IF bEnable THEN
	// Alarm_0420	420	Error	Blokada podnośnika lub brak zasilania - sprawdź czujnik lub odblokuj mechanicznie
	//Error 1 - podnośnik nie porusza się pomimo wysterowania 
	tonErrorHeightChange(IN:=(bHeightMotorUp OR bHeightMotorDown) AND nLastPositionHeightCV=lrHeightMotorCV, PT:=T#3S);
	IF tonErrorHeightChange.Q THEN
		IF NOT arfbAlarm[0].bActive THEN
			bHeightMotorUp:=FALSE;
			bHeightMotorDown:=FALSE;
			arfbAlarm[0].Raise(nTimeStamp:=0);
		END_IF
	ELSE	
		IF  arfbAlarm[0].bActive AND bReset THEN
			arfbAlarm[0].Clear(nTimeStamp:=0, bResetConfirmation:= FALSE);
		END_IF	
// 		bHeightMotorUp:=FALSE;
// 		bHeightMotorDown:=FALSE;
// 		bError := TRUE;
// 		nErrorNr:=241;
// 		//nErrorNr := nErrorNr+iStationIndex;
// 		sErrorDescription:='Blokada podnośnika lub brak zasilania - sprawdź czujnik lub odblokuj mechanicznie';	
	END_IF
	// Alarm_0421	421	Error	Wartość zadana wysokości jest większa od maksymalnej - zmień ustawienia w recepturze {0}
	//Error 7 - Bład nastaw max
	tonMaxHeight(IN:=nPositionHeightSV>lrMaxHeight AND NOT bHomingDone AND eState=E_Station.eStarting,PT:=T#0S);
	IF tonMaxHeight.Q THEN
		arfbAlarm[1].ipArguments.Clear() .AddLReal(lrMaxHeight);
		IF NOT arfbAlarm[1].bActive THEN
			bHeightMotorUp:=FALSE;
			bHeightMotorDown:=FALSE;
			arfbAlarm[1].Raise(nTimeStamp:=0);
		END_IF
	ELSE	
		IF  arfbAlarm[1].bActive AND bReset THEN
			arfbAlarm[1].Clear(nTimeStamp:=0, bResetConfirmation:= FALSE);
		END_IF	
// 		bHeightMotorUp:=FALSE;
// 		bHeightMotorDown:=FALSE;
// 		bError := TRUE;
// 		nErrorNr:=242;
// 		//nErrorNr := nErrorNr+iStationIndex;
// 		sErrorDescription:='Wartość zadana wysokości jest większa od maksymalnej - zmień ustawienia w recepturze';
// 		sErrorDescription2:=REAL_TO_STRING(LREAL_TO_INT(lrMaxHeight));
	END_IF
	// Alarm_0422	422	Error	Wartość zadana wysokości jest mniejsza od minimalnej - zmień ustawienia w recepturze {0}
	//Error 8 - Bład nastaw min
tonMinHeight(IN:=nPositionHeightSV<lrMinHeight AND NOT bHomingDone AND eState=E_Station.eStarting,PT:=T#0S);
IF tonMinHeight.Q AND NOT bStateError THEN
	arfbAlarm[2].ipArguments.Clear() .AddLReal(lrMinHeight);
		IF NOT arfbAlarm[2].bActive THEN
			bHeightMotorUp:=FALSE;
			bHeightMotorDown:=FALSE;
			arfbAlarm[2].Raise(nTimeStamp:=0);
		END_IF
	ELSE	
		IF  arfbAlarm[2].bActive AND bReset THEN
			arfbAlarm[2].Clear(nTimeStamp:=0, bResetConfirmation:= FALSE);
		END_IF	
	//	bHeightMotorUp:=FALSE;
	//	bHeightMotorDown:=FALSE;
	//	bError := TRUE;
	//	nErrorNr:=243;
	//	//nErrorNr := nErrorNr+iStationIndex;
	//	sErrorDescription:='Wartość zadana wysokości jest mniejsza od minimalnej - zmień ustawienia w recepturze';
	//	sErrorDescription2:=REAL_TO_STRING(LREAL_TO_INT(lrMinHeight));	
END_IF

ELSE
	bError := FALSE;
END_IF

	
//******************PRZEJŚCIE DO eERROR*****************************

IF bError AND NOT bStateError THEN
	IF eLastState = eRunning THEN
		bCycleNotDone := TRUE;
	END_IF
	eState := E_Station.eError;
END_IF

//****************WYŚWIETLANIE STATUSU BLEDU***********************

(*Wyświetlanie błedu na wyjściu*)
bError							:= FALSE;
FOR nAlarmNumerator := 0 TO 19 DO
	bError						:= bError OR arfbAlarm[nAlarmNumerator].bActive;
END_FOR

(*Przepisywanie nazwy stacji*)
sErrorStationName := WSTRING_TO_STRING(sStationName);

//Jezeli nie zbazowane to potrzebne bazowanie
IF NOT bHeightMotorEncoderHomed  THEN
	bHomingDone:=FALSE;
END_IF
END_ACTION

ACTION HeightMotor:
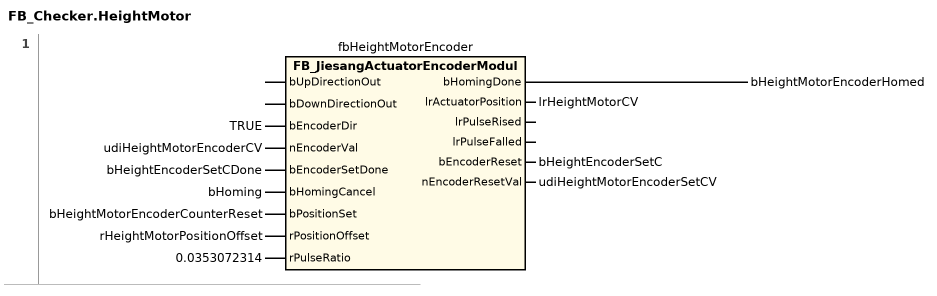
// NETWORK 1
fbHeightMotorEncoder(
    bEncoderDir := TRUE,
    nEncoderVal := udiHeightMotorEncoderCV,
    bEncoderSetDone := bHeightEncoderSetCDone,
    bHomingCancel := bHoming,
    bPositionSet := bHeightMotorEncoderCounterReset,
    rPositionOffset := rHeightMotorPositionOffset,
    rPulseRatio := 0.0353072314,
    lrActuatorPosition => lrHeightMotorCV,
    bEncoderReset => bHeightEncoderSetC,
    nEncoderResetVal => udiHeightMotorEncoderSetCV); // FB_JiesangActuatorEncoderModul
bHeightMotorEncoderHomed := fbHeightMotorEncoder.bHomingDone;
END_ACTION

ACTION Homing:
//BAZOWANIE

tofHeightMotorDown(IN:=bHeightMotorDown, PT:=T#1S); //Zabezpieczenie przed zbyt szybkim przełączeniem pomiędzy Down a Up, bezpiecznieki sie palą
	
//Podnoszenie stacji do maksymalnej pozycji
IF NOT bHeightMotorEncoderHomed OR rtEncoderHomed.Q THEN
	bHeightMotorUp:=(*TRUE*) NOT tofHeightMotorDown.Q;;
	bHeightMotorDown:=FALSE;
	IF tonHeightNoChange.Q THEN
		bHeightMotorEncoderCounterReset:=TRUE;
		bHeightMotorUp:=FALSE;
    END_IF
	//Jesli enkoder zbazowany zakończ bazowanie	
	IF rtEncoderHomed.Q THEN
		bHeightMotorUp:=FALSE;
		bHeightMotorDown:=FALSE;
		eState:=E_Station.eHomingDone;
	END_IF		
		
//Po podniesieniu stacji opuszczanie do ustalonej wysokości
ELSIF bHeightMotorEncoderHomed THEN
	bHeightMotorEncoderCounterReset:=FALSE;
	bHeightMotorUp:=lrHeightMotorCV<=nPositionHeightSV;
	bHeightMotorDown:=lrHeightMotorCV>=nPositionHeightSV;
	//Kiedy stacja osiągnie wysokość zadaną
	IF ABS(lrHeightMotorCV-nPositionHeightSV)<0.4 OR tonLimitPosMaxReachedDelay.Q OR tonLimitPosMinReachedDelay.Q THEN
		bHeightMotorDown:=FALSE;
		bHeightMotorUp:=FALSE;
		eState:=E_Station.eHomingDone;
	END_IF			
END_IF
END_ACTION

ACTION ManualMovements:

//W trybie ruchów manualnych wykonuj ruchy za pomocą rozkazów manualnych
IF NOT bRun THEN
	
	bHeightMotorUp:=bManualHeightMotorUp;
	bHeightMotorDown:=bManualHeightMotorDown;
ELSE	//Kasuje zeby po cyklu nic sie nie poruszało

	bManualHeightMotorUp  := FALSE;
	bManualHeightMotorDown  := FALSE;
END_IF


IF bHoming OR bHeightSet THEN
	eState:=E_Station.eHoming;
END_IF
	
Running();
	
//Zabezpieczenie przed kolizją stacji poprzez ruch podnośnika	
IF bHeightMotorDown AND lrHeightMotorCV<=lrMinHeight AND NOT bHoming AND NOT bHeightSet THEN
	bHeightMotorDown:=FALSE;
END_IF	

IF bHeightMotorUp AND lrHeightMotorCV>=lrMaxHeight AND NOT bHoming AND NOT bHeightSet THEN
	bHeightMotorUp:=FALSE;
END_IF
END_ACTION

ACTION Running:

//Timery
tofMotorUpPermition(IN:=bHeightMotorDown,PT:=T#250MS);
tofMotorDownPermition(IN:=bHeightMotorUp ,PT:=T#250MS);
tonOutputState(IN:=eRunningState=E_CheckerState.eFormPresent OR
				eRunningState=E_CheckerState.eBottleOK  OR
				eRunningState=E_CheckerState.eLidOK	 OR
				eRunningState=E_CheckerState.eCapOK OR
				eRunningState=E_CheckerState.eCapNOK
				,PT:=T#10MS);

CASE eRunningState OF
	
	E_CheckerState.eDisabled:
			eRunningState:=E_CheckerState.eReady;

	
	//SPRAWDZANIEGOTOWY DO PRACY
	E_CheckerState.eReady:
		//Jeśli wykryto czujnik formatki przejdź do stanu zasysania platynki
		IF bFormSensor THEN
			eRunningState:=E_CheckerState.eFormPresent;	
		END_IF

	//WYKRYTO FORMATKĘ
	E_CheckerState.eFormPresent:
		//Wykryto formatkę
		IF bBottleSensor THEN
			eRunningState:=E_CheckerState.eBottleOK;
		ELSIF bLidSensor THEN
			eRunningState:=E_CheckerState.eLidOK;
		ELSIF NOT bWenglorSensor THEN
			IF bCapSensor THEN
				eRunningState:=E_CheckerState.eCapOK;
			END_IF
		ELSIF bWenglorSensor THEN
			IF	bWenglorCapOk THEN
				eRunningState:=E_CheckerState.eCapOK;
			END_IF	
		ELSIF bCapNOKSensor THEN
			eRunningState:=E_CheckerState.eCapNOK;
		END_IF
		IF NOT bFormSensor THEN
			eRunningState:=E_CheckerState.eReady;
		END_IF

	//BUTELKA W FORMATCE
	E_CheckerState.eBottleOK:
		IF NOT bFormSensor THEN
			eRunningState:=E_CheckerState.eReady;
		END_IF
	
	//PLATYNKA OK
	E_CheckerState.eLidOK:
		IF NOT bFormSensor THEN
			eRunningState:=E_CheckerState.eReady;
		END_IF
	
	//NASADKA OK
	E_CheckerState.eCapOK:
		IF bCapNOKSensor THEN
			eRunningState:=E_CheckerState.eCapNOK;
		END_IF
		IF NOT bFormSensor THEN
			eRunningState:=E_CheckerState.eReady;
		END_IF	
		
		
	//NASADKA NOK
	E_CheckerState.eCapNOK:
		IF NOT bFormSensor THEN
			eRunningState:=E_CheckerState.eReady;
		END_IF			

END_CASE
END_ACTION

ACTION Statistics:

rtrigCycleTimerRead(CLK:=eRunningState=E_CheckerState.eFormPresent);
IF rtrigCycleTimerRead.Q THEN
		tCycleTime:=tonCycleTimer.ET;
END_IF
tonCycleTimer(IN:=eState>E_Station.eReady,PT:=T#1D);
END_ACTION

END_FUNCTION_BLOCK

// ---- POUs/FB/FB_VisionChecker_new.TcPOU
(*
Nazwa:			FB_VisionChecker
Opis:			stacja sprawdzania platynek czujnikiem wizyjnym
Wersja:			v1.0
Data:			2023-05-30
Autor:			DP
Urzadzenia:		Czujnik wizyjny KEYENCE
Konfiguracja:	
Info:
- 
*)

FUNCTION_BLOCK FB_VisionChecker_new
VAR_INPUT
	bEnable:BOOL;				//Zezowlenie na pracę stacji sprawdzania
	bEStop:BOOL;				//Stop Awaryjny nieaktywny
	bRun:BOOL;					//Rozkaz łapania 	
	bHoming:BOOL;				//Zezwolenie na wykonanie bazowania i pozycjonowania stacji sprawdzania
//	bHeightSet:BOOL;			//Ustaw wysokość
	bIgnoreError:BOOL;			//Ignorowania błędów cyklu pracy
	bReset:BOOL;				//Reset błędu, jeśli w stanie "eError"
//	nPositionHeightSV:LREAL;	//Wysokość zadana na której ma znajdować się stacja sprawdzania
	bManualMovement:BOOL; 		//Uruchomienie trybu ruchów ręcznych
//	lrMaxHeight:LREAL;			//Maksymalna wysokość stacji sprawdzania
//	lrMinHeight:LREAL;			//Minimalna wysokość stacji sprawdzania
	uiCameraActualProgram:UINT;
	iCameraSetProgram:INT;
	bCameraError:BOOL; 
	bCameraGood:BOOL; 	
	bCameraLogic1CapPresent:BOOL; 		
	bCameraBusy:BOOL; 	
	//StepMode
//	bStepMode				: BOOL;		//Włączony tryb skokowy sterowania podnośnikami (tylko w serwisie)
//	lrSetPosStepMode		: LREAL; 	//Ruch podnośnika o zadaną wartość w trybie krokowym (tylko w serwisie)
	
//	_HEIGHTMOTOR_ :BOOL;	
//	bHeightMotorEncoderPulse :BOOL;			//Sygnał impulsów enkodera siłownika
//	rHeightMotorPositionOffset :REAL;		//Wysokość bazowani podnośnika

	_ALARMINFO_ :BOOL;
	iStationIndex:UDINT;					//Numer stacji 
	sStationName:STRING;					//Nazwa stacji	

END_VAR
VAR_OUTPUT	
	eState: E_Station;						//Stan ogólny bloku
	eRunningState: E_CheckerState;			//Stan stacji sprawdzania
	bError: BOOL;							//Błąd stacji
	nErrorNr: UDINT;						//Nr błędu stacji sprawdzania
	sErrorDescription:STRING(200);			//Opis błędu
	sErrorDescription2:STRING(200);			//Opis błędu
	sErrorStationName:STRING;				//Nazwa stacji
	udiStationID: UDINT;				// Nr stacji

//	bHeightMotorUp:BOOL;					//Sterowanie silnikiem podnośnika  - RUCH W GÓRĘ
//	bHeightMotorDown:BOOL;					//Sterowanie silnikiem podnośnika  - RUCH W DÓŁ
//	lrHeightMotorCV:LREAL;					//Aktualna wysokość stacji sprawdzania
	bCameraTrigger:BOOL; 
	uiCameraProgram:UINT; 
	bCameraChangeProgram:BOOL; 	
	bCheckOK:BOOL;							//Platynka OK
	bCapPresent:BOOL;
	tCycleTime:TIME;	
	bHomingDone:BOOL;						//Wymagane ponowne bazowanie (blad podczas bazowania lub stop awaryjny)
	bCycleDone:BOOL;
	bCycleNotDone:BOOL;
	AsProgramDescription: ARRAY [0..10] OF STRING;	// Opis programów

END_VAR
VAR
//	tonHeightNoChange: TON; // Timer wykrycia braku ruchu siłownika zmiany wysokości stacji
//	nLastPositionHeightCV: LREAL;// Pozycja podnośnika w poprzednim cyklu programu
//	tonErrorHeightChange: TON; // Timer błędu podnośnika
	rtEncoderHomed:R_TRIG;
	tonCycleTimer:TON;
	rtrigCycleTimerRead:R_TRIG;
	tonTriggerDelay: TON;
	tonNotBusyDelay: TON;
	tonLidNOK: TON;
	tofMotorUpPermition: TOF;
	tofMotorDownPermition: TOF;
	tonLimitPosMinReachedDelay: TON;
	tonLimitPosMaxReachedDelay: TON;
	tonMaxHeight: TON;
	tonMinHeight: TON;
	
	//Podnośnik Jiesang	
	fbHeightMotorEncoder: FB_JiesangActuatorEncoder_1;	// Blok enkodera podnośnika chwytaka stabilizującego pod zakręcarką	
	bHeightMotorEncoderCounterReset:BOOL; 				// Sygnał resetu enkodera
	bHeightMotorEncoderHomed:BOOL;						// Informacja od enkodera że jest zbazowany

	eLastState: E_Station;								// Stan ogólny bloku
	eLastRunningState: E_CheckerState;					// Stan podbloku
	eLastStateTemp: E_Station;							// Stan ogólny bloku
	eLastRunningStateTemp: E_CheckerState;				// Stan podbloku	
	
	bStateError: BOOL;

	//Step Mode
	rtStepModeUp			: R_TRIG;
	rtStepModeDown			: R_TRIG;
	lrStepModeHeightMotorSV	: LREAL;
	bStepModeMoving			: BOOL;
	tofStepModeMoving		: TOF;	
	rtCheckingEnd			: R_TRIG;
	tonbCameraChangeProgram: TON;
	rtuiCameraActualProgram: R_TRIG;
	tonTryChangeProgram: TON;
END_VAR

//HeightMotor();
ErrorHandling();
Control();
Statistics();
Programs();
aStationID();

(*Zapisywanie ostatniego stanu*)
IF eLastStateTemp<>eState THEN
	eLastState := eLastStateTemp;
END_IF
eLastStateTemp := eState;
IF eLastRunningStateTemp<>eRunningState THEN
	eLastRunningState := eLastRunningStateTemp;
END_IF
eLastRunningStateTemp := eRunningState;
(*Koniec Zapisywanie ostatniego stanu*)

//nLastPositionHeightCV:=lrHeightMotorCV;

ACTION aStationID:
udiStationID	:=	iStationIndex;
END_ACTION

ACTION Control:

	(** TIMERY**)
	rtEncoderHomed				(CLK:=bHeightMotorEncoderHomed,																Q=>);


	(*****Wyłączenie enable*****)
	IF NOT bEnable THEN
		IF eState <> E_Station.eDisabled AND eState <> E_Station.ePreparingToDisable THEN
				eState 							:=	E_Station.ePreparingToDisable; 
		END_IF	
	END_IF

	(*****Estop*****)
	IF NOT bEstop  THEN	
		IF eState <> E_Station.eAborted AND eState <> E_Station.eAborting AND eState <> E_Station.eDisabled THEN
				eState 							:=	E_Station.eAborting; 
		END_IF
	END_IF

	
	CASE eState OF
	/////////////////////////////	
		E_Station.eDisabled: 					// Stan nieaktywnosci (Stacja wyłączona) 
		
			IF bEnable THEN
				eState 							:=	E_Station.ePreparingToReady; 
			END_IF 
			
    /////////////////////////////	    
		E_Station.eAborted: 					// Stan bezpiecznego zatrzymania (po Abortingu) 

			IF bEStop THEN
				eState 							:=	E_Station.ePreparingToReady;
			END_IF
			
	/////////////////////////////	
		E_Station.eAborting:                 	// Stan bezpiecznego zatrzymywania (po EStopie)
			
//			bHeightMotorUp						:=	FALSE;
//			bHeightMotorDown					:=	FALSE;
			eState 								:=	E_Station.eAborted;  
			eRunningState						:=	E_CheckerState.eDisabled;
			
	/////////////////////////////			
		E_Station.eError:                 	 	// Stan błędu 	
	
			IF bReset THEN
				eState 							:=	E_Station.eResetting;
			ELSE
				ResetCommands();
			END_IF
			
	/////////////////////////////
		E_Station.eResetting:					// Stan resetowania bledu (po Errorze)
			
			bError := FALSE;
			IF NOT bError THEN
				nErrorNr 						:=	0;
   				sErrorDescription 				:=	'';
				eState 							:=	E_Station.ePreparingToReady;
			ELSE
				eState 							:=	E_Station.eError;
			END_IF
        
	/////////////////////////////
		E_Station.eManualMovement:     			// Stan ruchów manualnych  
       
			ManualMovements();
			//Wyjście z trybu serwisowego
//			IF NOT bManualMovement THEN
//				bHeightMotorUp					:=	FALSE;
//				bHeightMotorDown				:=	FALSE;	
//				eState							:=	E_Station.eReady;
//			END_IF

	/////////////////////////////
		E_Station.eHoming:						// Stan bazowania 

			Homing();
//			IF NOT bHoming AND NOT bHeightSet THEN
//				bHeightMotorDown				:=	FALSE;
//				bHeightMotorUp					:=	FALSE;
				eState							:=	E_Station.ePreparingToReady;
//			END_IF		
			
	/////////////////////////////
		E_Station.eHomingDone:                  // Stan wykonania bazowania 
		
//			bHeightMotorDown					:=	FALSE;
//			bHeightMotorUp						:=	FALSE;
//			bHeightMotorEncoderCounterReset		:=	FALSE;
			bHomingDone							:=	TRUE;
//			IF NOT bHoming AND NOT bHeightSet THEN
			   eState							:=	E_Station.eReady;
//			END_IF
			
	/////////////////////////////
		E_Station.ePreparingToReady:            // Stan przygotowywania do gotowosci (zawsze przed Ready)  
		
			eRunningState						:=	E_CheckerState.eReady;
			eState								:=	E_Station.eReady;	
			
	/////////////////////////////
		E_Station.ePreparingToDisable:          // Stan przygotowywania do nieaktywnosci (po wyłączeniu Enable) 
  
//			bHeightMotorUp						:=	TRUE;
//			bHeightMotorDown					:=	FALSE;	
//			IF tonHeightNoChange.Q THEN
//				bHeightMotorUp					:=	FALSE;
				eState							:=	E_Station.eDisabled;
				eRunningState					:=	E_CheckerState.eDisabled;
//			END_IF	
				
	/////////////////////////////
		E_Station.eReady:						// Stan gotowosci 
			
			IF bRun AND NOT bCycleDone AND NOT bCycleNotDone THEN
				eState 							:=	E_Station.eStarting; 
			END_IF
			IF bHoming (*OR bHeightSet*) THEN
				eState 							:=	E_Station.eHoming; 
			END_IF
			IF bManualMovement THEN
				//Jeśli przejście w tryb ruchów manualnych przepisz wszystkie stany siłowników sterowanych przez moduł
				//aby zapobiec ewentualnym kolizjom po wejściu w tryb serwisowy
//				bManualHeightMotorUp			:=	bHeightMotorUp;
//				bManualHeightMotorDown			:=	bHeightMotorDown;
				eState 							:=	E_Station.eManualMovement; 
			END_IF
			IF NOT bRun THEN
				bCycleDone 						:=	FALSE;
				bCycleNotDone 					:=	FALSE;			
			END_IF
			
	/////////////////////////////
		E_Station.eStopping:					// Stan zatrzymywania 
			
			Running();
			bCameraTrigger						:= FALSE;
			bCheckOK							:= FALSE;
			eState								:=	E_Station.eReady;
			
	/////////////////////////////
		E_Station.eStarting:                  	// Stan uruchamiania (po Ready)
		
			eRunningState						:= E_CheckerState.eReady;
			eState								:= E_Station.eRunning; 

	/////////////////////////////
		E_Station.eRunning:               		// Stan wykonywania cyklu (po Startingu), w tym stanie osobny
 
			Running();
			IF NOT bRun THEN 					(*Przerywanie cyklu*)
				eState							:=	E_Station.eStopping;
				bCycleNotDone					:=	TRUE;
			END_IF
			(*IF bCycleDone OR bCycleNotDone THEN (*Cykl zakończony*)
				eState 				 := E_Station.eReady;
			END_IF*)						
			
	/////////////////////////////		
	END_CASE
END_ACTION

ACTION ErrorHandling:
//OBSŁUGA BŁĘDÓW STACJI SPRAWDZANIA

//************LISTA BŁĘDÓW***************
bStateError:= (eState=E_Station.eError) OR (eState=E_Station.eResetting) OR bIgnoreError;

IF bEnable THEN

//	//Error 1 - podnośnik nie porusza się pomimo wysterowania 
//	tonErrorHeightChange(IN:=(bHeightMotorUp OR bHeightMotorDown) AND nLastPositionHeightCV=lrHeightMotorCV, PT:=T#3S);
//	IF tonErrorHeightChange.Q AND NOT bStateError THEN
//		bHeightMotorUp:=FALSE;
//		bHeightMotorDown:=FALSE;
//		bError := TRUE;
//		nErrorNr:=301;
//		//nErrorNr := nErrorNr+iStationIndex;
//		sErrorDescription:='Blokada podnośnika lub brak zasilania - sprawdź czujnik lub odblokuj mechanicznie';	
//	END_IF
	
//	//Error 2 - Bład nastaw max
//	tonMaxHeight(IN:=nPositionHeightSV>lrMaxHeight AND NOT bHomingDone AND eState=E_Station.eStarting,PT:=T#0S);
//	IF tonMaxHeight.Q AND NOT bStateError THEN
//		bHeightMotorUp:=FALSE;
//		bHeightMotorDown:=FALSE;
//		bError := TRUE;
//		nErrorNr:=302;
//		//nErrorNr := nErrorNr+iStationIndex;
//		sErrorDescription:='Wartość zadana wysokości jest większa od maksymalnej - zmień ustawienia w recepturze';
//		sErrorDescription2:=REAL_TO_STRING(LREAL_TO_INT(lrMaxHeight));
//	END_IF
	
	//Error 3 - Bład nastaw min
	//tonMinHeight(IN:=nPositionHeightSV<lrMinHeight AND NOT bHomingDone AND eState=E_Station.eStarting,PT:=T#0S);
	//IF tonMinHeight.Q AND NOT bStateError THEN
	//	bHeightMotorUp:=FALSE;
	//	bHeightMotorDown:=FALSE;
	//	bError := TRUE;
	//	nErrorNr:=303;
	//	//nErrorNr := nErrorNr+iStationIndex;
	//	sErrorDescription:='Wartość zadana wysokości jest mniejsza od minimalnej - zmień ustawienia w recepturze';
	//	sErrorDescription2:=REAL_TO_STRING(LREAL_TO_INT(lrMinHeight));	
	//END_IF

ELSE
	bError := FALSE;
END_IF

	
//******************PRZEJŚCIE DO eERROR*****************************

IF bError AND NOT bStateError THEN
	IF eLastState = eRunning THEN
		bCycleNotDone := TRUE;
	END_IF
	eState := E_Station.eError;
END_IF

//****************WYŚWIETLANIE STATUSU BLEDU***********************

(*Wyświetlanie błedu na wyjściu*)
bError;

(*Przepisywanie nazwy stacji*)
sErrorStationName := sStationName;

//Jezeli nie zbazowane to potrzebne bazowanie
IF NOT bHeightMotorEncoderHomed  THEN
	bHomingDone:=FALSE;
END_IF
END_ACTION

ACTION Homing:
//BAZOWANIE
eState:=E_Station.eHomingDone;
	
////Podnoszenie stacji do maksymalnej pozycji
//IF NOT bHeightMotorEncoderHomed OR rtEncoderHomed.Q THEN
//	bHeightMotorUp:=TRUE;
//	bHeightMotorDown:=FALSE;
//	IF tonHeightNoChange.Q THEN
//		bHeightMotorEncoderCounterReset:=TRUE;
//		bHeightMotorUp:=FALSE;
//    END_IF
//	//Jesli enkoder zbazowany zakończ bazowanie	
//	IF rtEncoderHomed.Q THEN
//		bHeightMotorUp:=FALSE;
//		bHeightMotorDown:=FALSE;
//		eState:=E_Station.eHomingDone;
//	END_IF		
		
////Po podniesieniu stacji opuszczanie do ustalonej wysokości
//ELSIF bHeightMotorEncoderHomed THEN
//	bHeightMotorEncoderCounterReset:=FALSE;
//	bHeightMotorUp:=lrHeightMotorCV<=nPositionHeightSV;
//	bHeightMotorDown:=lrHeightMotorCV>=nPositionHeightSV;
//	//Kiedy stacja osiągnie wysokość zadaną
//	IF ABS(lrHeightMotorCV-nPositionHeightSV)<1 OR tonLimitPosMaxReachedDelay.Q OR tonLimitPosMinReachedDelay.Q THEN
//		bHeightMotorDown:=FALSE;
//		bHeightMotorUp:=FALSE;
//		eState:=E_Station.eHomingDone;
//	END_IF			
//END_IF
END_ACTION

ACTION ManualMovements:

//W trybie ruchów manualnych wykonuj ruchy za pomocą rozkazów manualnych
IF NOT bRun THEN
	eRunningState		:=	E_CheckerState.eReady;
	bCameraTrigger		:=	FALSE;
	bCheckOK			:=	FALSE;
//	bHeightMotorUp		:=	bManualHeightMotorUp;
//	bHeightMotorDown	:=	bManualHeightMotorDown;
ELSE	//Kasuje zeby po cyklu nic sie nie poruszało
//	bManualHeightMotorUp  := FALSE;
//	bManualHeightMotorDown  := FALSE;
END_IF


IF bHoming (*OR bHeightSet*) THEN
	eState:=E_Station.eHoming;
END_IF
	
Running();

	
//Zabezpieczenie przed kolizją stacji poprzez ruch podnośnika	
//IF bHeightMotorDown AND lrHeightMotorCV<=lrMinHeight AND NOT bHoming AND NOT bHeightSet THEN
//	bHeightMotorDown:=FALSE;
//END_IF	

//IF bHeightMotorUp AND lrHeightMotorCV>=lrMaxHeight AND NOT bHoming AND NOT bHeightSet THEN
//	bHeightMotorUp:=FALSE;
//END_IF
END_ACTION

ACTION Programs:
tonbCameraChangeProgram	(IN:=bCameraChangeProgram,PT:=T#1S);
tonTryChangeProgram	(IN:=uiCameraActualProgram <> uiCameraProgram AND NOT bCameraChangeProgram, PT:=T#5S);
rtuiCameraActualProgram	(CLK:=uiCameraActualProgram <> uiCameraProgram,	Q=>);
uiCameraProgram	:=	INT_TO_UINT(iCameraSetProgram);

IF rtuiCameraActualProgram.Q	 OR  tonTryChangeProgram.Q THEN
	bCameraChangeProgram	:=	TRUE;
END_IF
IF tonbCameraChangeProgram.Q THEN
	bCameraChangeProgram	:=	FALSE;
END_IF

(*Narzędzia*)
AsProgramDescription[0] := '1. opak:butelka płaska, nasadka:wbijana biała';
AsProgramDescription[1] := '2. opak:rezerwa, nasadka:rezerwa';
AsProgramDescription[2] := '3. opak:rezerwa, nasadka:rezerwa';
AsProgramDescription[3] := '4. opak:rezerwa, nasadka:rezerwa';
AsProgramDescription[4] := '5. opak:rezerwa, nasadka:rezerwa';
AsProgramDescription[5] := '6. opak:rezerwa, nasadka:rezerwa';
AsProgramDescription[6] := '7. opak:rezerwa, nasadka:rezerwa';
AsProgramDescription[7] := '8. opak:rezerwa, nasadka:rezerwa';
AsProgramDescription[8] := '9. opak:rezerwa, nasadka:rezerwa';
AsProgramDescription[9] := '10. opak:rezerwa, nasadka:rezerwa';
AsProgramDescription[10] := '11. opak:rezerwa, nasadka:rezerwa';
END_ACTION

ACTION ResetCommands:

//bStepModeMoving 			:= FALSE;
//bHeightMotorDown			:= FALSE;
//bHeightMotorUp				:= FALSE;
//bManualHeightMotorUp		:= FALSE;
//bManualHeightMotorDown		:= FALSE;
END_ACTION

ACTION Running:

//Timery
//tofMotorUpPermition		(IN:=	bHeightMotorDown,								PT:=T#250MS);
//tofMotorDownPermition	(IN:=	bHeightMotorUp,									PT:=T#250MS);
tonTriggerDelay			(IN:=	eRunningState=E_CheckerState.eFormPresent,		PT:=T#50MS);//bylo 50
tonNotBusyDelay			(IN:=	tonTriggerDelay.Q AND NOT bCameraBusy,
																				PT:=T#50MS);
tonLidNOK				(IN:=	eRunningState=E_CheckerState.eFormPresent,
																				PT:=T#50MS);				

CASE eRunningState OF
	
	E_CheckerState.eDisabled:
	
		eRunningState		:=	E_CheckerState.eReady;
	
	//SPRAWDZANIEGOTOWY DO PRACY
	E_CheckerState.eReady:
		
		IF bRun THEN
			eRunningState	:=	E_CheckerState.eFormPresent;	
		END_IF

	//WYKRYTO SLOIK
	E_CheckerState.eFormPresent:
	
		bCameraTrigger		:= TRUE;
		IF	tonTriggerDelay.Q THEN
			IF tonNotBusyDelay.Q AND bCameraGood THEN
				eRunningState	:=	E_CheckerState.eLidOK;		
			ELSIF tonNotBusyDelay.Q  THEN
				eRunningState	:=	E_CheckerState.eLidNOK;	
			END_IF	
		END_IF
		
	
	//BUTELKA W FORMATCE
	E_CheckerState.eBottleOK:
	;
	
	//PLATYNKA OK
	E_CheckerState.eLidOK:
	
		bCheckOK	:= TRUE;
		bCycleDone	:= TRUE;
		bCapPresent	:= bCameraLogic1CapPresent;	
	
	//PLATYNKA NOK
	E_CheckerState.eLidNOK:

		bCheckOK	:= FALSE;	
		bCycleDone	:= TRUE;
		bCapPresent	:= bCameraLogic1CapPresent;
		
	//NASADKA OK
	E_CheckerState.eCapOK:
	;
		
	//NASADKA NOK
	E_CheckerState.eCapNOK:
	;		

	E_CheckerState.eChecking:
	;
		
END_CASE
END_ACTION

ACTION Statistics:

rtrigCycleTimerRead(CLK:=eRunningState=E_CheckerState.eLidOK OR eRunningState=E_CheckerState.eLidNOK);
IF rtrigCycleTimerRead.Q THEN
		tCycleTime:=tonCycleTimer.ET;
END_IF
tonCycleTimer(IN:=eState>E_Station.eReady,PT:=T#1D);
END_ACTION

END_FUNCTION_BLOCK

// ---- POUs/FB/Various/FB_Average.TcPOU
(********************************************************************************************)
(*							Beckhoff Automation Poland										*)
(*								FB_Average	 v1.2											*)
(*									2.02.2011												*)
(*								v1.2 Optymalizacja wewnętrzna								*)
(*					Blok funkcyjny obliczający średnią z wartości wejściowej rValue			*)
(*					w zadanym przedziale czasowym lub z określonej ilości pomiarów			*)
(*__________________________________________________________________________________________*)
FUNCTION_BLOCK FB_Average
VAR_INPUT
	rValue : 			REAL;			(*Uśredniana wartość*)
	tInterval : 		TIME;			(*Co jaki czas ma byc robiony wpis*)
END_VAR
VAR_OUTPUT
	rAverage: 			REAL; 			(*Wartość średnia*)
END_VAR
VAR CONSTANT
	MAX_INDEX: 			USINT 	:= 10 ;	(*Ilość wpisów do uśredniania*)
END_VAR
VAR
	aData: 				ARRAY[0..MAX_INDEX] OF REAL;
	nIndex:		 		USINT;			(*Ostatni wpis, czyli przyjmuje wartosci od 0 do MAX_INDEX - 1*)
	i:					USINT;			(*Iterator*)
	ttimer: 			TON;
	suma: 				REAL;
END_VAR

ttimer(IN:= NOT ttimer.Q, PT:= tInterval, Q=> , ET=> );

IF nIndex = 0 THEN	(*Na poczatku wypelniamy pierwsza komorke w tablicy*)
	nIndex := 1;
	aData[0] := rValue;
END_IF

IF ttimer.Q THEN
	suma := 0;
	FOR i := 1 TO nIndex DO
		aData[i - 1] := aData[i];
		suma := suma + aData[i];
	END_FOR
	IF	nIndex < (MAX_INDEX) THEN
		nIndex := nIndex + 1;
	END_IF
	aData[nIndex] := rValue;
END_IF

rAverage := suma/nIndex;

END_FUNCTION_BLOCK

// ---- POUs/P09_CapPuttedCheck.TcPOU
(*
Nazwa:			P09_CapPuttedCheck
Opis:			Stacja sprawdzania nasadek
Wersja:			v0.1
Data:			2018-10-10
Autor:			DP
Urzadzenia:		
Konfiguracja:	
Info:

*)
PROGRAM P09_CapPuttedCheck
VAR_INPUT
	IbCapPuttedCheckSensor 				AT %I*		:BOOL;		// Wejście wykrycia nasadki 
	IbCapPuttedCheckFormSensor 			AT %I*		:BOOL;		// Wejście wykrycia formatek w sprawdzaniu nasadek
END_VAR
VAR
	fbCapPuttedCheck								:FB_Checker;
	eCapPuttedCheckState							:E_Station; 			// Stan pracy podajnika platynek			
	eCapPuttedCheckRunningState						:E_CheckerState; 		// Stan pracy podajnika platynek
	fbCapPuttedCheckState							:FB_State;
	
	IbCapPuttedCheckHeightEncoderPulses				AT %I*:BOOL;		//	(*PLC.A14*) 	// Enkoder podnośnika czujnika kontroli nakrętki
	QbCapPuttedCheckHeightUpCmd 					AT %Q*: BOOL; 				//	(*PLC.A19*) 	// Wyjście sterujące podnośnikiem sprawdzania nasadek w formatkach, Silnik w górę
	QbCapPuttedCheckHeightDownCmd 					AT %Q*: BOOL; 			//	(*PLC.A19*)		// Wyjście sterujące podnośnikiem sprawdzania nasadek w formatkach, Silnik w dół
	IbCapPuttedCheckWenglorFormSensor				AT %I*:BOOL;
	fbIbCapPuttedCheckFormSensor					:FB_InputFilter; //Wejście przefiltrowane czujnika

	IbCapPuttedCheckEncoderSetCDone				AT %I*: BOOL;	
    IudiCapPuttedCheckHeightEncoderCV          AT %I*: UDINT;
    QbCapPuttedCheckHeightEncoderSetC 			AT %Q*: BOOL;
    QudiCapPuttedCheckHeightEncoderSetCV       AT %Q*: UDINT;
	
	TimerCapPuttedCheckEnable						: TOF;
	tonCapPuttedCheckEnable							: TON;		
	rtEnable										: R_TRIG;
	tonCapPuttedFormsCheckRFID						: TON;
	rtCapPuttedFormCheck							: R_TRIG;

	tonStoppingCapPuttedTooLong: TON;
	IdiCapPuttedCheckSensorCV_Wenglor					AT %I*:DINT;
	IbCapPuttedCheckSensorScale_Wenglor					AT %I*:BYTE;
	IbCapPuttedCheckSensorWarning_1_Wenglor				AT %I*:BOOL;
	IbCapPuttedCheckSensorWarning_2_Wenglor				AT %I*:BOOL;	
	IbCapPuttedCheckSensorWarning_3_Wenglor				AT %I*:BOOL;
	IbCapPuttedCheckSensorWarning_4_Wenglor				AT %I*:BOOL;
	IbCapPuttedCheckSensorWarning_Wenglor				AT %I*:BOOL;
	IbCapPuttedCheckSensorError_Wenglor                	AT %I*:BOOL;
	IbCapPuttedCheckSensorSSC1_Wenglor                 	AT %I*:BOOL;
	IbCapPuttedCheckSensorSSC2_Wenglor                 	AT %I*:BOOL;
	QbCapPuttedCheckSensorControlSignal_Wenglor			AT %Q*:BOOL;
	QbCapPuttedCheckSensorFindMe_Wenglor				AT %Q*:BOOL;
	QbCapPuttedCheckSensorTeachSSC1_Wenglor             AT %Q*:BOOL;
	QbCapPuttedCheckSensorTeachSSC2_Wenglor				AT %Q*:BOOL;
	
	bCapPuttedCheckSensorWenglorBottleTooFar	:BOOL;
	bCapPuttedCheckSensorWenglorBottleTooClose	:BOOL;
	bCapPuttedCheckSensorWenglorNoData	:BOOL;
	diDistanceSensorToTransporter		:DINT;
	
	
	lrCapPuttedCheckSensorCV						: LREAL;
	lrCapPuttedCheckSensorFilteredCV				: LREAL;
	lrCapPuttedCheckSensorAveragedCV				: LREAL;	
	fbCapPuttedCheckSensorFilter					: FB_FilterEx;
	fbCapPuttedCheckSensorAverage					: FB_Average;	
	lrCapPuttedCheckSensorLimitLow: LREAL;
	lrCapPuttedCheckSensorLimitHigh: LREAL;
	bCapPuttedCheckSensorLimitOK: BOOL;
	bCapPuttedCheckSensorLimitNOK: BOOL;	
	tonCapPuttedCheckSensorLimitOK: TON;
	tonCapPuttedCheckSensorLimitNOK: TON;
	bCapPuttedCheckSensorShinyMode: BOOL;
	bCapPuttedCheckSensorPointedMode: BOOL;	
END_VAR



tonStoppingCapPuttedTooLong(IN:=P00_PackML.fbPMLAuto.ePMLState = E_PMLState.ePMLState_STOPPING,PT:=T#3S);
IF P00_PackML.fbPMLAuto.ePMLState = E_PMLState.ePMLState_EXECUTE OR P00_PackML.fbPMLAuto.ePMLState = E_PMLState.ePMLState_STARTING THEN
	bCapPuttedCheckRun:=TRUE;
ELSIF tonStoppingCapPuttedTooLong.Q THEN
	bCapPuttedCheckRun:=FALSE;
END_IF
aCapPuttedCheck();
aCapPuttedCheckSensor();

tonCapPuttedFormsCheckRFID(IN:=IbCapPuttedCheckFormSensor, PT:=T#25MS);//było 10
rtCapPuttedFormCheck(CLK:=tonCapPuttedFormsCheckRFID.Q);


fbIbCapPuttedCheckFormSensor(bIN:=IbCapPuttedCheckFormSensor, tFilterTimeOn:=T#10MS, tFilterTimeOff:=T#10MS);

(* BAZOWANIE - ZMIAN*)
tonCapPuttedCheckEnable(IN:=fbCapPuttedCheck.bEnable,PT:=T#5S); (*Dodany ton bo Wizka zjebnie wgrywa zmienne, najpierw włacza Enabla a potem dopiero wybiera recepture*)
rtEnable(CLK:=tonCapPuttedCheckEnable.Q,Q=>);

IF rtEnable.Q AND (P00_PackML.fbPMLAuto.ePMLState = E_PMLState.ePMLState_IDLE OR P00_PackML.fbPMLAuto.ePMLState = E_PMLState.ePMLState_EXECUTE)  THEN
		VIS.bCapPuttedCheckHeightSet											:= TRUE;
ELSIF fbCapPuttedCheck.eState=E_Station.eHomingDone  OR VIS.bErrorOccure THEN
 		VIS.bCapPuttedCheckHeightSet											:= FALSE;
END_IF

(*KONIEC BAZOWANIE - ZMIANA*)

(********* GENEROWANIE STANU STACJI DO WIZKI**********)
fbCapPuttedCheckState(
	eState																		:= eCapPuttedCheckState , 
	bRun																		:= P00_PackML.fbPMLAuto.ePMLState = E_PMLState.ePMLState_EXECUTE ,	
	eCheckerRunningState														:= eCapPuttedCheckRunningState , 
	sStateDesc																	=> VIS.sCapPuttedCheckState,
	iState																		=> VIS.iCapPuttedCheckState );
(***** KONIEC GENEROWANIE STANU STACJI DO WIZKI*******)	

(*Opoznienie wyłączanie enabla*)
TimerCapPuttedCheckEnable (IN:=bCapPuttedCheckEnable , PT:=T#2S);



(****WENGLOR*************)
lrCapPuttedCheckSensorLimitLow:=diDistanceSensorToTransporter-VIS.iPackageHeightShow;
lrCapPuttedCheckSensorLimitHigh:=diDistanceSensorToTransporter-VIS.iPackageHeightShow+150;

ACTION aCapPuttedCheck:
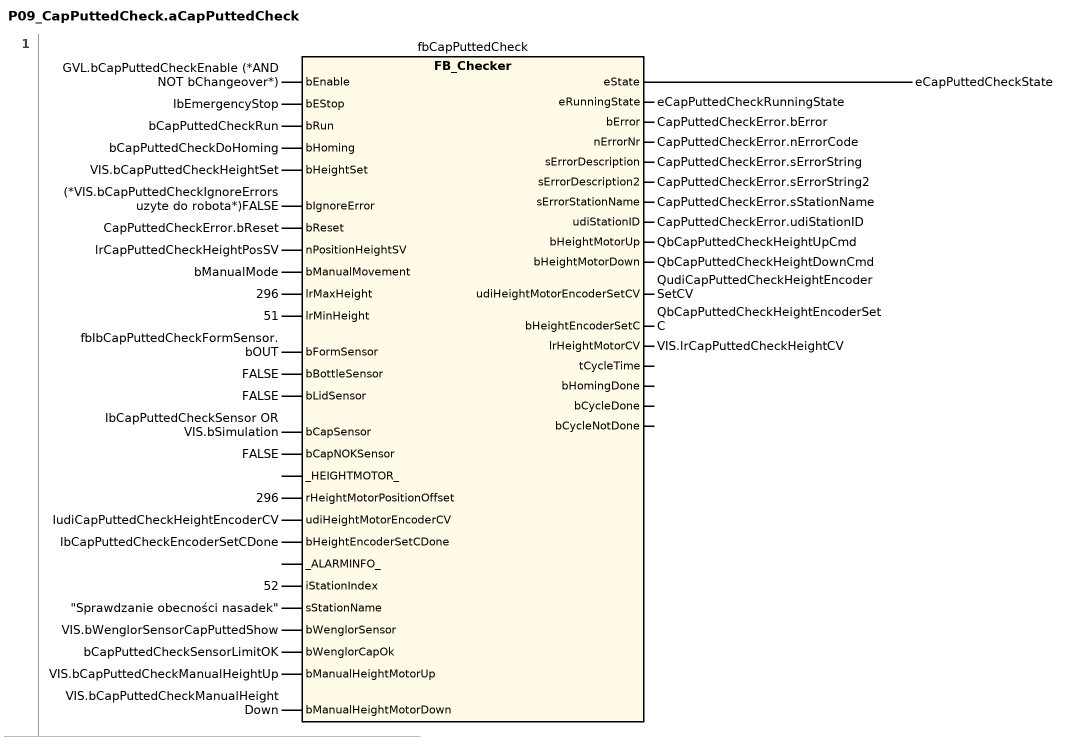
// NETWORK 1
fbCapPuttedCheck(
    bEnable := GVL.bCapPuttedCheckEnable (*AND NOT bChangeover*),
    bEStop := IbEmergencyStop,
    bRun := bCapPuttedCheckRun,
    bHoming := bCapPuttedCheckDoHoming,
    bHeightSet := VIS.bCapPuttedCheckHeightSet,
    bIgnoreError := (*VIS.bCapPuttedCheckIgnoreErrors uzyte do robota*)FALSE,
    bReset := CapPuttedCheckError.bReset,
    nPositionHeightSV := lrCapPuttedCheckHeightPosSV,
    bManualMovement := bManualMode,
    lrMaxHeight := 296,
    lrMinHeight := 51,
    bFormSensor := fbIbCapPuttedCheckFormSensor.bOUT,
    bBottleSensor := FALSE,
    bLidSensor := FALSE,
    bCapSensor := IbCapPuttedCheckSensor OR VIS.bSimulation,
    bCapNOKSensor := FALSE,
    rHeightMotorPositionOffset := 296,
    udiHeightMotorEncoderCV := IudiCapPuttedCheckHeightEncoderCV,
    bHeightEncoderSetCDone := IbCapPuttedCheckEncoderSetCDone,
    iStationIndex := 52,
    sStationName := "Sprawdzanie obecności nasadek",
    bWenglorSensor := VIS.bWenglorSensorCapPuttedShow,
    bWenglorCapOk := bCapPuttedCheckSensorLimitOK,
    bManualHeightMotorUp := VIS.bCapPuttedCheckManualHeightUp,
    bManualHeightMotorDown := VIS.bCapPuttedCheckManualHeightDown,
    eRunningState => eCapPuttedCheckRunningState,
    bError => CapPuttedCheckError.bError,
    nErrorNr => CapPuttedCheckError.nErrorCode,
    sErrorDescription => CapPuttedCheckError.sErrorString,
    sErrorDescription2 => CapPuttedCheckError.sErrorString2,
    sErrorStationName => CapPuttedCheckError.sStationName,
    udiStationID => CapPuttedCheckError.udiStationID,
    bHeightMotorUp => QbCapPuttedCheckHeightUpCmd,
    bHeightMotorDown => QbCapPuttedCheckHeightDownCmd,
    udiHeightMotorEncoderSetCV => QudiCapPuttedCheckHeightEncoderSetCV,
    bHeightEncoderSetC => QbCapPuttedCheckHeightEncoderSetC,
    lrHeightMotorCV => VIS.lrCapPuttedCheckHeightCV); // FB_Checker
eCapPuttedCheckState := fbCapPuttedCheck.eState;
END_ACTION

ACTION aCapPuttedCheckSensor:
(*
Nazwa:			P09_CapPuttedCheck.aCapPuttedCheckSensor
Opis:			Dalmierz
Wersja:			v0.1
Data:			2024-12-30
Autor:			DP
Urzadzenia:		
Konfiguracja:	
Info:
- testy dalmierza, filtrowanie

*)

IF IdiCapPuttedCheckSensorCV_Wenglor < 2_000_000 THEN
	lrCapPuttedCheckSensorCV	:=	DINT_TO_LREAL(ABS(IdiCapPuttedCheckSensorCV_Wenglor))/1000.0;
END_IF

IF IdiCapPuttedCheckSensorCV_Wenglor =-2147483640 THEN
	bCapPuttedCheckSensorWenglorBottleTooClose:=TRUE;
ELSIF IdiCapPuttedCheckSensorCV_Wenglor = 2147483640 THEN
	bCapPuttedCheckSensorWenglorBottleTooFar:=TRUE;
ELSE
	bCapPuttedCheckSensorWenglorBottleTooClose:=FALSE;
	bCapPuttedCheckSensorWenglorBottleTooFar:=FALSE;
END_IF

IF IdiCapPuttedCheckSensorCV_Wenglor=2147483644 THEN
	bCapPuttedCheckSensorWenglorNoData:=TRUE;
ELSE
	bCapPuttedCheckSensorWenglorNoData:=FALSE;
END_IF 

fbCapPuttedCheckSensorFilter(
							rIn:=				LREAL_TO_REAL(lrCapPuttedCheckSensorCV), 
							tTimeConstant:= 	T#9MS, 
							rOut=>				lrCapPuttedCheckSensorFilteredCV);
				

fbCapPuttedCheckSensorAverage(
							rValue:=			LREAL_TO_REAL(lrCapPuttedCheckSensorCV),
							tInterval:=			T#3MS,
							rAverage=>			lrCapPuttedCheckSensorAveragedCV);
							
IF vis.bWenglorSensorCapModeShow =0 THEN
	bCapPuttedCheckSensorShinyMode:=FALSE;
	bCapPuttedCheckSensorPointedMode:=FALSE;
ELSIF vis.bWenglorSensorCapModeShow =1 THEN
	bCapPuttedCheckSensorShinyMode:=TRUE;
	bCapPuttedCheckSensorPointedMode:=FALSE;
ELSIF vis.bWenglorSensorCapModeShow =2 THEN
	bCapPuttedCheckSensorShinyMode:=FALSE;
	bCapPuttedCheckSensorPointedMode:=TRUE;		
END_IF


							
lrCapPuttedCheckSensorLimitLow;
lrCapPuttedCheckSensorLimitHigh;
IF bCapPuttedCheckRun THEN
IF NOT bCapPuttedCheckSensorShinyMode AND NOT bCapPuttedCheckSensorPointedMode THEN	

	VIS.iPackageCapTypeShow			;// Typ nasadki (0-Fliptop, 1-Pompka/Atomizer, 2-Kulka, 3-Airless, 4-, 5- Deko, 6-Nakrętka_słoika
	IF VIS.iPackageCapTypeShow	= 6 THEN
		(*sloik*)		tonCapPuttedCheckSensorLimitOK	(IN:=(lrCapPuttedCheckSensorFilteredCV > VIS.iPackageHeightShow), PT:=T#200MS);
	ELSE
		(*nie sloik*)	tonCapPuttedCheckSensorLimitOK	(IN:=(lrCapPuttedCheckSensorFilteredCV > VIS.iPackageHeightShow), PT:=T#20MS);
	END_IF
	IF  IbCapPuttedCheckFormSensor AND tonCapPuttedCheckSensorLimitOK.Q THEN
		bCapPuttedCheckSensorLimitOK	:=	TRUE;
	ELSIF (*NOT IbCapPuttedCheckFormSensor*)P00_ReadRFIDCard.fbBeforeScrewerReader.bCodeReaded OR P00_ReadRFIDCard.fbBeforeScrewerReader.bError OR vis.bCycleReset THEN
		bCapPuttedCheckSensorLimitOK	:=	FALSE;	
	END_IF
	tonCapPuttedCheckSensorLimitNOK	(IN:=(lrCapPuttedCheckSensorFilteredCV > lrCapPuttedCheckSensorLimitHigh), PT:=T#20MS);
	
	IF IbCapPuttedCheckFormSensor AND tonCapPuttedCheckSensorLimitNOK.Q THEN
		bCapPuttedCheckSensorLimitNOK	:=	TRUE;
	ELSE
		bCapPuttedCheckSensorLimitNOK	:=	FALSE;	
	END_IF
ELSIF bCapPuttedCheckSensorPointedMode THEN	
	(* W przypadku szpiczastych nakrętek  lepszy jest sygnał nie filtrowany

	*)
	tonCapPuttedCheckSensorLimitOK	(IN:=(lrCapPuttedCheckSensorCV > VIS.iPackageHeightShow), PT:=T#10MS);
	IF IbCapPuttedCheckFormSensor(*IbCapPuttedCheckWenglorFormSensor*) AND tonCapPuttedCheckSensorLimitOK.Q THEN
		bCapPuttedCheckSensorLimitOK	:=	TRUE;
	ELSE
		bCapPuttedCheckSensorLimitOK	:=	FALSE;	
	END_IF
	tonCapPuttedCheckSensorLimitNOK	(IN:=(lrCapPuttedCheckSensorCV > lrCapPuttedCheckSensorLimitHigh), PT:=T#10MS);
	
	IF IbCapPuttedCheckFormSensor AND tonCapPuttedCheckSensorLimitNOK.Q THEN
		bCapPuttedCheckSensorLimitNOK	:=	TRUE;
	ELSE
		bCapPuttedCheckSensorLimitNOK	:=	FALSE;	
	END_IF		
ELSE		
	(* W przypadku błyszczących nakrętek od słoika lepszy jest sygnał nie filtrowany
		ciężko dobrać czasówke NOK, może powinna być w nastawach
	*)
	tonCapPuttedCheckSensorLimitOK	(IN:=(lrCapPuttedCheckSensorCV > VIS.iPackageHeightShow+20) , PT:=T#20MS);
	IF IbCapPuttedCheckFormSensor AND tonCapPuttedCheckSensorLimitOK.Q THEN
		bCapPuttedCheckSensorLimitOK	:=	TRUE;
	ELSE
		bCapPuttedCheckSensorLimitOK	:=	FALSE;	
	END_IF
	tonCapPuttedCheckSensorLimitNOK	(IN:=(lrCapPuttedCheckSensorCV > lrCapPuttedCheckSensorLimitHigh), PT:=T#50MS);
	
	IF IbCapPuttedCheckFormSensor AND tonCapPuttedCheckSensorLimitNOK.Q THEN
		bCapPuttedCheckSensorLimitNOK	:=	TRUE;
	ELSE
		bCapPuttedCheckSensorLimitNOK	:=	FALSE;	
	END_IF	
END_IF	
END_IF


//Logika Vasyl
VIS.iPackageHeightShow; //wartość wysokości formatki z butelką
VIS.iPackageCappedHeightShow;
IdiCapPuttedCheckSensorCV_Wenglor; //pomiar do powierzchni
diDistanceSensorToTransporter:=615; //pomiar od transportera do powierzchni transportera
END_ACTION

END_PROGRAM

// ---- POUs/P06_WickFeeder.TcPOU
PROGRAM P06_WickFeeder
VAR_INPUT
	IbWickFeederDragHomingSensor 			  	: BOOL;				// Czujnik bazowania
	IbWickFeederDragUpSensor 			 	  	: BOOL;				// Czujnik
	IbWickFeederDragDownSensor 				 	: BOOL;				// Czujnik
	IbWickFeederDragLeadBefore1UpSensor 		: BOOL;				// Czujnik
	IbWickFeederDownSensor1 					: BOOL;								
	IbWheelLevelSensor								: BOOL;			

	IbWheelSensor									: BOOL;			//Czujnik zapełnienia rękawa
	IbQueFullAfterWheelSensor						: BOOL;			
	IbQueFullSensor									: BOOL;			//Czujnik zapełnienia rękawa
	IbWickAtPipe									: BOOL;			//Czujnik na końcu rękawa
	IbSeparatorPos1									: BOOL;			//Separator nad torem 1
	IbSeparatorPos2									: BOOL;			//Separator nad torem 2
	IbQueFullAtSleve1								: BOOL;			//Czujnik zapełnienia rękawa 1
	IbQueFullAtSleve2								: BOOL;			//Czujnik zapełnienia rękawa 2
	IbWickAtSleve1									: BOOL;			//Czujnik na końcu rękawa 1
	IbWickAtSleve2									: BOOL;			//Czujnik na końcu rękawa 2
	IbSleve1SeparatorOut							: BOOL;			//Separator nad butelką
	IbSleve2SeparatorOut							: BOOL;			//Separator nad butelką
	IbHammer1Up										: BOOL;			//Wbijak pozycja górna
	IbHammer1Down									: BOOL;			//Wbijak pozycja dolna
	IbHammer2Up										: BOOL;			//Wbijak pozycja górna
	IbHammer2Down									: BOOL;			//Wbijak pozycja dolna
	IbFormPositioningHide1							: BOOL; 
	IbFormPositioningHide2							: BOOL;

	QbStopper1										: BOOL;			//Stoper przed separatorem
	QbStopper2										: BOOL;			//Stoper przed separatorem
	QbSeparator1									: BOOL;			//Separator nad torem 1
	QbSeparator2									: BOOL;			//Separator nad torem 2
	QbSleve1SeparatorActIn							: BOOL;			//Separator pod rękawem
	QbSleve1SeparatorActOut							: BOOL;			//Separator nad butelką
	QbSleve2SeparatorActIn							: BOOL;			//Separator pod rękawem
	QbSleve2SeparatorActOut							: BOOL;			//Separator nad butelką
	QbHammer1										: BOOL;			//Wbijak 
	QbHammer2										: BOOL;			//Wbijak
	QbBlow1											: BOOL;
	QbSleeveBlow									: BOOL;
	QbFormPositioning								: BOOL;  		


	bMovetoEndPositionWickFeeder				: BOOL;	
	QbWickFeederDragActuator                  	: BOOL;				// Siłownikiem przeciągania (1 faza)					

	
	QbWickFeederSorterEngine					AT %Q*	: BOOL; 					// Wyjście silnikiem sortera
	QbWickFeederSorterAir 						AT %Q*	: BOOL; 					// Wyjście sterujące szybkim zaworem wydmuchu
	QbWickFeederSorterAir2 						AT %Q*	: BOOL; 					// Wyjście sterujące szybkim zaworem wydmuchu
	
	IbFuseWickFeederSorterEngineOK			AT %I*	: BOOL;					//Bezpiecznik silnika sortera OK

	QnWickFeederSorterVelocitySV 			AT %Q*	: UDINT; 		// Nastawa prędkości
	InWickFeederSorterVelocityCV 			AT %I*	: UDINT;		
	InWickFeederSorterSTW 					AT %I*	: UINT; 		// Statusword transportera wejściowo wyjściowego
	QnWickFeederSorterCTW 					AT %Q*	: UINT;  		// Controlword transportera we/wy
                                                  		
	TimerWickFeederSorterEnable						: TOF;
	tonWickFeederSorterEnable						: TON;
	
END_VAR
VAR
	//Podajnik knotów
	fbWickFeederSt									: FB_WickFeederStation; 				// Blok sterowania
	eWickFeederState								: E_Station; 							// Stan pracy podajnika platynek			
	eWickFeederRunningState							: E_WickFeederState; 					// Stan pracy podajnika platynek
	fbWickFeederState								: FB_State; 


	QbWickFeeder_HeightMotorUp 				AT %Q*	: BOOL;									// Sterowanie silnikiem podnosnika stacji w górę 
	QbWickFeeder_HeightMotorDown 			AT %Q*	: BOOL;									//Sterowanie silnikiem podnosnika stacji w dół
	
	
	IbWickFeeder2DownSensor1 				AT %I*	: BOOL;								
	IbWickFeederHeightEncoderSetCDone		AT %I*	: BOOL;	
	IudiWickFeederHeightEncoderCV         	AT %I*	: UDINT; 	
	QbWickFeederHeightEncoderSetC 			AT %Q*	: BOOL;		
	QudiWickFeederHeightEncoderSetCV       	AT %Q*	: UDINT; 	
	
	tofWickFeederEnable								: TOF;
	tonWickFeederEnable								: TON;
	rtEnable										: R_TRIG;

	bSimulation										: BOOL;
	
	bWickFeederWarning1								: BOOL;
	bWickFeederWarning2								: BOOL;
	
	//PRZECIAGANIE
	eWickFeederDragStation							: E_Station;
	eWickFeederDragRunningStation					: E_DragStationState;
	fbWickFeederDragStation							: FB_FormsDragStepper;

	tofWickFeederDragStationEnable					: TOF;	
	
	//WEJSCIA I WYJSCIA SPRZETOWE
	QbWickFeederDragLeadBefore1Actuator        		: BOOL;				// Siłownikiem prowadzenia przed 1(1 faza)
	QbWickFeederDragLeadBefore2Actuator        		: BOOL;				// Siłownikiem prowadzenia przed 1(1 faza)
	


	bTestManual										: BOOL;	
	bWickFeederSorterRunTest						: BOOL;
	bWickFeeder1RunTest								: BOOL;
	bWickFeeder2RunTest								: BOOL;
	tonQbSleve1SeparatorActIn						:TON;
	tonQbSleve2SeparatorActIn						:TON;	
END_VAR


ACT_Limits();
ACT_WickFeederStation();
ACT_WickFeederDragStation();
aWickFeederWarnings();

//GENEROWANIE STANU STACJI DO WIZKI
tonQbSleve1SeparatorActIn	(IN:=QbSleve1SeparatorActIn, PT:=T#100MS);
tonQbSleve2SeparatorActIn	(IN:=QbSleve2SeparatorActIn, PT:=T#100MS);

(* BAZOWANIE - ZMIAN*)
tonWickFeederEnable(IN := fbWickFeederSt.bEnable, PT := T#2S); (*Dodany ton bo Wizka zjebnie wgrywa zmienne, najpierw włacza Enabla a potem dopiero wybiera recepture*)
rtEnable(CLK := tonWickFeederEnable.Q, Q=>);
IF rtEnable.Q AND (P00_PackML.fbPMLAuto.ePMLState = Tc3_PackML.E_PMLState.ePMLState_IDLE OR 
   P00_PackML.fbPMLAuto.ePMLState = Tc3_PackML.E_PMLState.ePMLState_EXECUTE) THEN
    VIS.bWickFeederHeightSet 		:= TRUE;
ELSIF fbWickFeederst.eState = E_Station.eHomingDone OR VIS.bErrorOccure THEN
    VIS.bWickFeederHeightSet 		:= FALSE;
END_IF
(*KONIEC BAZOWANIE - ZMIANA*)

//PRZEPISYWANIE POMIARÓW

//SYMULACJA CZUJNIKÓW IGLIC

//Opoznienie wyłączanie enabla
tofWickFeederEnable(IN:= bWickFeederEnable, PT:=T#2S);

//KASOWANIE ROZKAZÓW CYKLI
IF fbWickFeederst.bCycleDone1 AND GVL.bManualMode THEN
	VIS.bWickFeeder1Run 			:= FALSE;
END_IF
IF fbWickFeederst.bCycleDone2 AND GVL.bManualMode THEN
	VIS.bWickFeeder2Run 			:= FALSE;
END_IF

IF bSimulation THEN
	IF fbWickFeederSt.eRunningState1 = E_WickFeederState.eReady  THEN
		VIS.bWickFeeder1Run	:= TRUE;
	END_IF
	IF fbWickFeederSt.eRunningState2 = E_WickFeederState.eReady  THEN
		VIS.bWickFeeder2Run	:= TRUE;
	END_IF	
	

	IF fbWickFeederSt.bCycleDone1 THEN		
		VIS.bWickFeeder1Run 		:= FALSE;	
	END_IF
	IF fbWickFeederSt.bCycleDone2 THEN		
		VIS.bWickFeeder2Run 		:= FALSE;	
	END_IF
END_IF

//Przeciąganie
tofWickFeederDragStationEnable(IN:= bWickFeederDragingStationEnable, PT:= T#2S);


////ZBIORNIK I SORTER KNOTÓW
aWickFeederSorterWarnings();
QbWickFeederSorterAir2 :=	QbWickFeederSorterEngine OR QbWickFeederSorterAir; //Dodatkowy przedmuch


(*Opoznienie wyłączanie enabla*)

ACTION ACT_Limits:
(*
Nazwa:			aSetRecipe
Opis:			Zapisywanie zmiennych gdy mają wartość 0 
Wersja:			v0.1
Data:			2022-06-22
Autor:			DP
Urzadzenia:		
Konfiguracja:	
Info:
- zabezpieczenie przed recepturami które nie mają tych parametrów i jest w nich wartość 0
*)

IF 	VIS.lrWickFeedingDragingStationStartPosition		= 0		THEN	VIS.lrWickFeedingDragingStationStartPosition		:=	8;		END_IF;
IF 	VIS.lrWickFeedingDragingStationEndPosition		= 0		THEN	VIS.lrWickFeedingDragingStationEndPosition		:=	138;	END_IF;
END_ACTION

ACTION ACT_WickFeederDragStation:
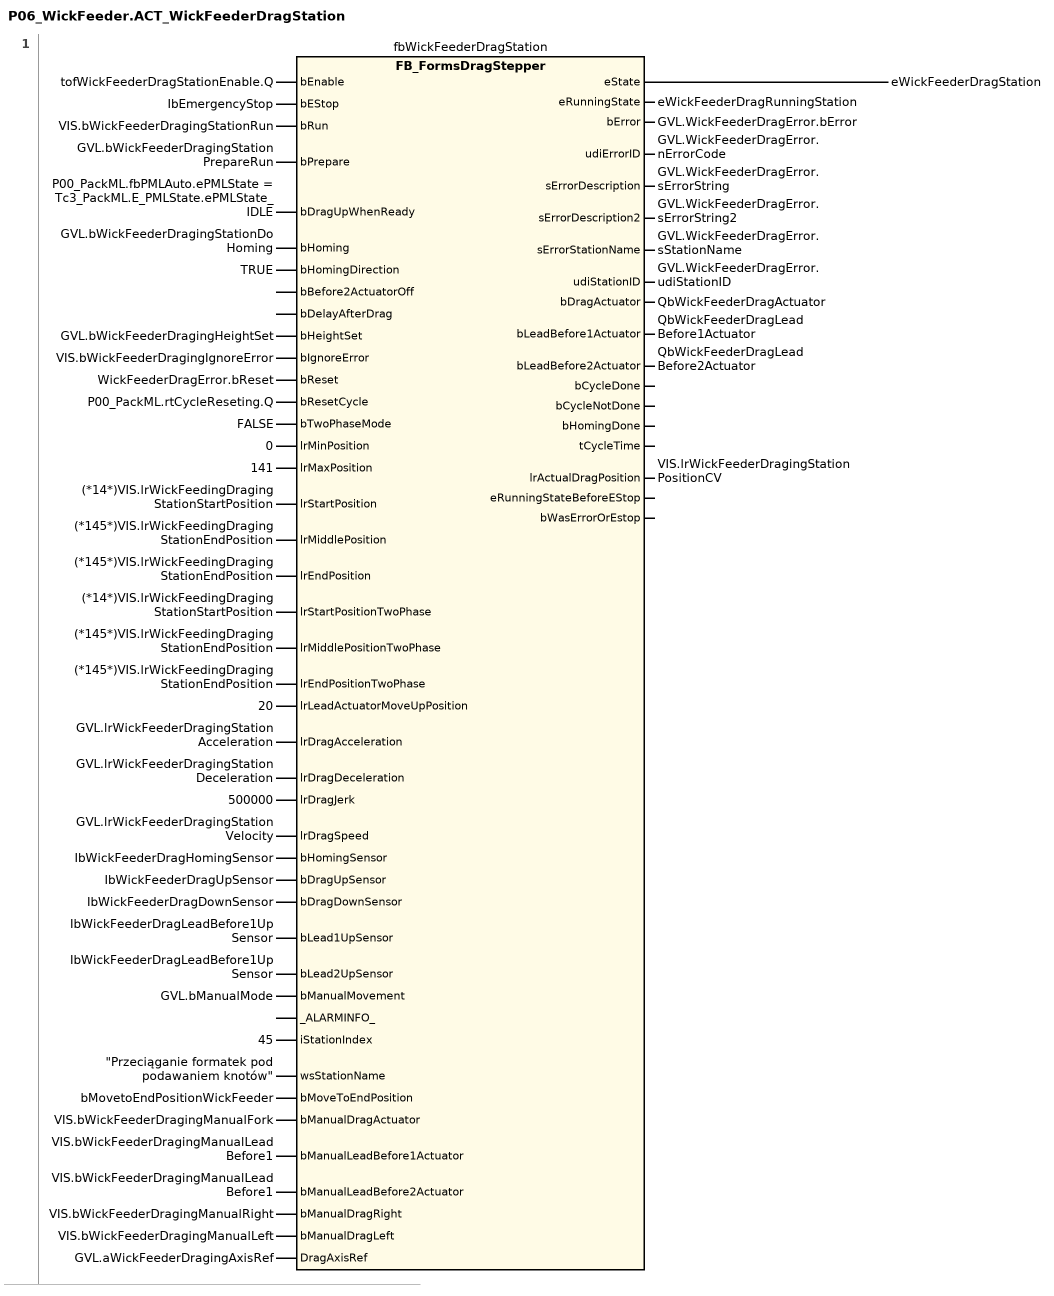
// NETWORK 1
fbWickFeederDragStation(
    bEnable := tofWickFeederDragStationEnable.Q,
    bEStop := IbEmergencyStop,
    bRun := VIS.bWickFeederDragingStationRun,
    bPrepare := GVL.bWickFeederDragingStationPrepareRun,
    bDragUpWhenReady := P00_PackML.fbPMLAuto.ePMLState = Tc3_PackML.E_PMLState.ePMLState_IDLE,
    bHoming := GVL.bWickFeederDragingStationDoHoming,
    bHomingDirection := TRUE,
    bHeightSet := GVL.bWickFeederDragingHeightSet,
    bIgnoreError := VIS.bWickFeederDragingIgnoreError,
    bReset := WickFeederDragError.bReset,
    bResetCycle := P00_PackML.rtCycleReseting.Q,
    bTwoPhaseMode := FALSE,
    lrMinPosition := 0,
    lrMaxPosition := 141,
    lrStartPosition := (*14*)VIS.lrWickFeedingDragingStationStartPosition,
    lrMiddlePosition := (*145*)VIS.lrWickFeedingDragingStationEndPosition,
    lrEndPosition := (*145*)VIS.lrWickFeedingDragingStationEndPosition,
    lrStartPositionTwoPhase := (*14*)VIS.lrWickFeedingDragingStationStartPosition,
    lrMiddlePositionTwoPhase := (*145*)VIS.lrWickFeedingDragingStationEndPosition,
    lrEndPositionTwoPhase := (*145*)VIS.lrWickFeedingDragingStationEndPosition,
    lrLeadActuatorMoveUpPosition := 20,
    lrDragAcceleration := GVL.lrWickFeederDragingStationAcceleration,
    lrDragDeceleration := GVL.lrWickFeederDragingStationDeceleration,
    lrDragJerk := 500000,
    lrDragSpeed := GVL.lrWickFeederDragingStationVelocity,
    bHomingSensor := IbWickFeederDragHomingSensor,
    bDragUpSensor := IbWickFeederDragUpSensor,
    bDragDownSensor := IbWickFeederDragDownSensor,
    bLead1UpSensor := IbWickFeederDragLeadBefore1UpSensor,
    bLead2UpSensor := IbWickFeederDragLeadBefore1UpSensor,
    bManualMovement := GVL.bManualMode,
    iStationIndex := 45,
    wsStationName := "Przeciąganie formatek pod podawaniem knotów",
    bMoveToEndPosition := bMovetoEndPositionWickFeeder,
    bManualDragActuator := VIS.bWickFeederDragingManualFork,
    bManualLeadBefore1Actuator := VIS.bWickFeederDragingManualLeadBefore1,
    bManualLeadBefore2Actuator := VIS.bWickFeederDragingManualLeadBefore1,
    bManualDragRight := VIS.bWickFeederDragingManualRight,
    bManualDragLeft := VIS.bWickFeederDragingManualLeft,
    DragAxisRef := GVL.aWickFeederDragingAxisRef,
    eRunningState => eWickFeederDragRunningStation,
    bError => GVL.WickFeederDragError.bError,
    udiErrorID => GVL.WickFeederDragError.nErrorCode,
    sErrorDescription => GVL.WickFeederDragError.sErrorString,
    sErrorDescription2 => GVL.WickFeederDragError.sErrorString2,
    sErrorStationName => GVL.WickFeederDragError.sStationName,
    udiStationID => GVL.WickFeederDragError.udiStationID,
    bDragActuator => QbWickFeederDragActuator,
    bLeadBefore1Actuator => QbWickFeederDragLeadBefore1Actuator,
    bLeadBefore2Actuator => QbWickFeederDragLeadBefore2Actuator,
    lrActualDragPosition => VIS.lrWickFeederDragingStationPositionCV); // FB_FormsDragStepper
eWickFeederDragStation := fbWickFeederDragStation.eState;
END_ACTION

ACTION ACT_WickFeederStation:
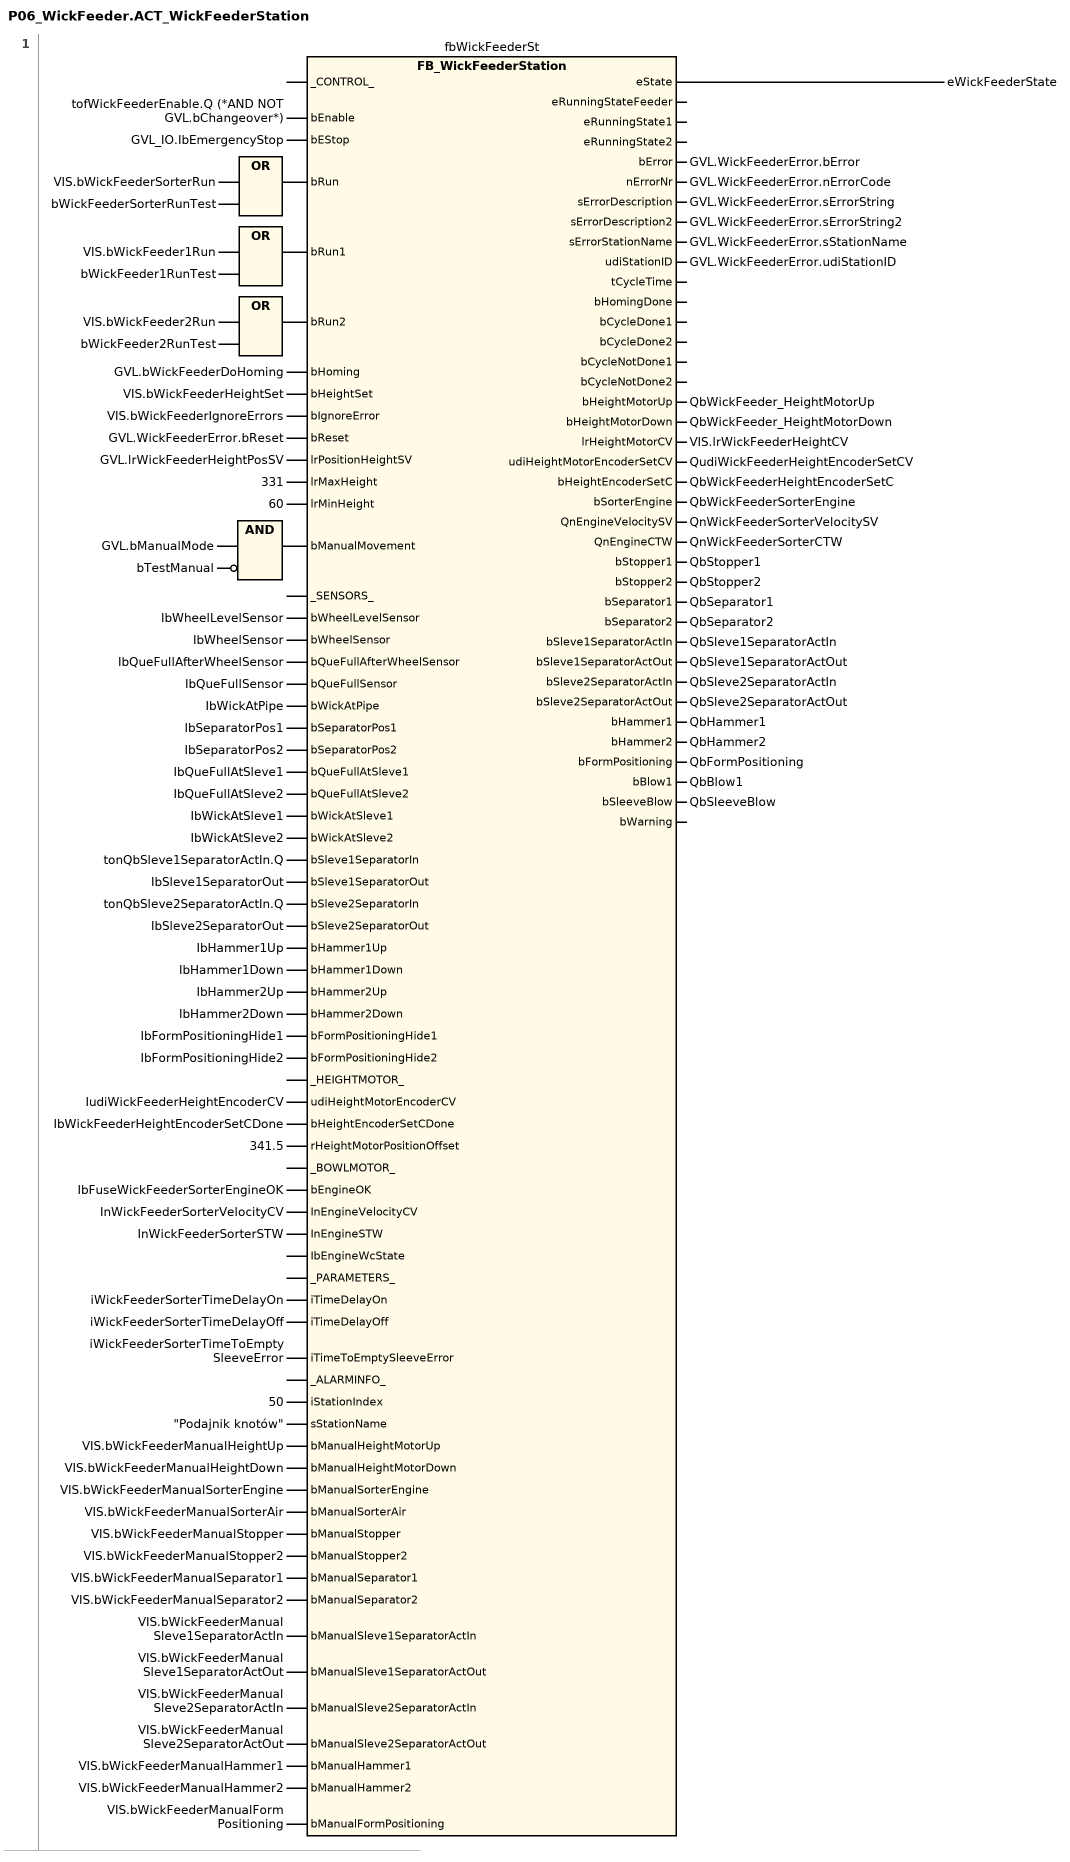
// NETWORK 1
fbWickFeederSt(
    bEnable := tofWickFeederEnable.Q (*AND NOT GVL.bChangeover*),
    bEStop := GVL_IO.IbEmergencyStop,
    bRun := VIS.bWickFeederSorterRun OR bWickFeederSorterRunTest,
    bRun1 := VIS.bWickFeeder1Run OR bWickFeeder1RunTest,
    bRun2 := VIS.bWickFeeder2Run OR bWickFeeder2RunTest,
    bHoming := GVL.bWickFeederDoHoming,
    bHeightSet := VIS.bWickFeederHeightSet,
    bIgnoreError := VIS.bWickFeederIgnoreErrors,
    bReset := GVL.WickFeederError.bReset,
    lrPositionHeightSV := GVL.lrWickFeederHeightPosSV,
    lrMaxHeight := 331,
    lrMinHeight := 60,
    bManualMovement := GVL.bManualMode AND NOT bTestManual,
    bWheelLevelSensor := IbWheelLevelSensor,
    bWheelSensor := IbWheelSensor,
    bQueFullAfterWheelSensor := IbQueFullAfterWheelSensor,
    bQueFullSensor := IbQueFullSensor,
    bWickAtPipe := IbWickAtPipe,
    bSeparatorPos1 := IbSeparatorPos1,
    bSeparatorPos2 := IbSeparatorPos2,
    bQueFullAtSleve1 := IbQueFullAtSleve1,
    bQueFullAtSleve2 := IbQueFullAtSleve2,
    bWickAtSleve1 := IbWickAtSleve1,
    bWickAtSleve2 := IbWickAtSleve2,
    bSleve1SeparatorIn := tonQbSleve1SeparatorActIn.Q,
    bSleve1SeparatorOut := IbSleve1SeparatorOut,
    bSleve2SeparatorIn := tonQbSleve2SeparatorActIn.Q,
    bSleve2SeparatorOut := IbSleve2SeparatorOut,
    bHammer1Up := IbHammer1Up,
    bHammer1Down := IbHammer1Down,
    bHammer2Up := IbHammer2Up,
    bHammer2Down := IbHammer2Down,
    bFormPositioningHide1 := IbFormPositioningHide1,
    bFormPositioningHide2 := IbFormPositioningHide2,
    udiHeightMotorEncoderCV := IudiWickFeederHeightEncoderCV,
    bHeightEncoderSetCDone := IbWickFeederHeightEncoderSetCDone,
    rHeightMotorPositionOffset := 341.5,
    bEngineOK := IbFuseWickFeederSorterEngineOK,
    InEngineVelocityCV := InWickFeederSorterVelocityCV,
    InEngineSTW := InWickFeederSorterSTW,
    iTimeDelayOn := iWickFeederSorterTimeDelayOn,
    iTimeDelayOff := iWickFeederSorterTimeDelayOff,
    iTimeToEmptySleeveError := iWickFeederSorterTimeToEmptySleeveError,
    iStationIndex := 50,
    sStationName := "Podajnik knotów",
    bManualHeightMotorUp := VIS.bWickFeederManualHeightUp,
    bManualHeightMotorDown := VIS.bWickFeederManualHeightDown,
    bManualSorterEngine := VIS.bWickFeederManualSorterEngine,
    bManualSorterAir := VIS.bWickFeederManualSorterAir,
    bManualStopper := VIS.bWickFeederManualStopper,
    bManualStopper2 := VIS.bWickFeederManualStopper2,
    bManualSeparator1 := VIS.bWickFeederManualSeparator1,
    bManualSeparator2 := VIS.bWickFeederManualSeparator2,
    bManualSleve1SeparatorActIn := VIS.bWickFeederManualSleve1SeparatorActIn,
    bManualSleve1SeparatorActOut := VIS.bWickFeederManualSleve1SeparatorActOut,
    bManualSleve2SeparatorActIn := VIS.bWickFeederManualSleve2SeparatorActIn,
    bManualSleve2SeparatorActOut := VIS.bWickFeederManualSleve2SeparatorActOut,
    bManualHammer1 := VIS.bWickFeederManualHammer1,
    bManualHammer2 := VIS.bWickFeederManualHammer2,
    bManualFormPositioning := VIS.bWickFeederManualFormPositioning,
    bError => GVL.WickFeederError.bError,
    nErrorNr => GVL.WickFeederError.nErrorCode,
    sErrorDescription => GVL.WickFeederError.sErrorString,
    sErrorDescription2 => GVL.WickFeederError.sErrorString2,
    sErrorStationName => GVL.WickFeederError.sStationName,
    udiStationID => GVL.WickFeederError.udiStationID,
    bHeightMotorUp => QbWickFeeder_HeightMotorUp,
    bHeightMotorDown => QbWickFeeder_HeightMotorDown,
    lrHeightMotorCV => VIS.lrWickFeederHeightCV,
    udiHeightMotorEncoderSetCV => QudiWickFeederHeightEncoderSetCV,
    bHeightEncoderSetC => QbWickFeederHeightEncoderSetC,
    bSorterEngine => QbWickFeederSorterEngine,
    QnEngineVelocitySV => QnWickFeederSorterVelocitySV,
    QnEngineCTW => QnWickFeederSorterCTW,
    bStopper1 => QbStopper1,
    bStopper2 => QbStopper2,
    bSeparator1 => QbSeparator1,
    bSeparator2 => QbSeparator2,
    bSleve1SeparatorActIn => QbSleve1SeparatorActIn,
    bSleve1SeparatorActOut => QbSleve1SeparatorActOut,
    bSleve2SeparatorActIn => QbSleve2SeparatorActIn,
    bSleve2SeparatorActOut => QbSleve2SeparatorActOut,
    bHammer1 => QbHammer1,
    bHammer2 => QbHammer2,
    bFormPositioning => QbFormPositioning,
    bBlow1 => QbBlow1,
    bSleeveBlow => QbSleeveBlow); // FB_WickFeederStation
eWickFeederState := fbWickFeederSt.eState;
END_ACTION

ACTION aWickFeederSorterWarnings:
// Sorter nasadek
(*
IF fbWickFeederSt.bWarning1 AND NOT WickFeederSorterWarning[0].bWarning THEN
	WickFeederSorterWarning[0].bWarning										:= TRUE;
	WickFeederSorterWarning[0].udiWarningCode									:= 33;	
	WickFeederSorterWarning[0].sDescription									:= 'Podajnik knotów | Niski poziom wkładów';
ELSIF NOT fbWickFeederSt.bWarning1  AND WickFeederSorterWarning[0].bAcknowledge THEN
	WickFeederSorterWarning[0].bWarning										:= FALSE;
	WickFeederSorterWarning[0].bAcknowledge									:= FALSE;
	VIS.uliWarningAcknowledge.14 										:= FALSE;
ELSIF WickFeederSorterWarning[0].bAcknowledge THEN
	WickFeederSorterWarning[0].bAcknowledge									:= TRUE;
END_IF*)
END_ACTION

ACTION aWickFeederWarnings:

//Warning 0
LidFeederWarning[0].sDescription:='Podajnik knotów | Niski poziom';
IF P06_WickFeeder.fbWickFeederSt.bWarning AND NOT LidFeederWarning[0].bWarning AND bWickFeederEnable THEN
	LidFeederWarning[0].bWarning:=TRUE;
ELSIF NOT P06_WickFeeder.fbWickFeederSt.bWarning  AND LidFeederWarning[0].bAcknowledge THEN
	LidFeederWarning[0].bWarning		:=	FALSE;
	LidFeederWarning[0].bAcknowledge	:=	FALSE;
	VIS.uliWarningOccure.39				:=	FALSE;
ELSIF LidFeederWarning[0].bAcknowledge THEN
	LidFeederWarning[0].bAcknowledge	:=	TRUE;
END_IF

//Warning 1
(*WickFeederWarning[1].sDescription:='Podajnik knotów 2 | Brak knotów w zasobniku';
IF bWickFeederWarning2 AND NOT WickFeederWarning[1].bWarning AND bWickFeederEnable THEN
	WickFeederWarning[1].bWarning:=TRUE;
ELSIF NOT bWickFeederWarning2 AND WickFeederWarning[1].bAcknowledge THEN
	WickFeederWarning[1].bWarning		:=	FALSE;
	WickFeederWarning[1].bAcknowledge	:=	FALSE;
	VIS.uliWarningOccure.40				:=	FALSE;
ELSIF WickFeederWarning[1].bAcknowledge THEN
	WickFeederWarning[1].bAcknowledge	:=	TRUE;
END_IF*)
END_ACTION

END_PROGRAM

// ---- POUs/FB/FB_WickFeederStation.TcPOU
(*
Nazwa:			FB_WickFeederStation
Opis:			Podajnik knotów
Wersja:			v1.0
Data:			2025-12-29
Autor:			MK
Urzadzenia:		Podnosnik stacji, grzałka, czujnik temp, ssawka
Konfiguracja:	
Info: 
*)




FUNCTION_BLOCK FB_WickFeederStation
VAR_INPUT
	_CONTROL_:BOOL;	
	bEnable:BOOL;					//Zezowlenie na pracę podajnika knotów
	bEStop:BOOL;					//Stop awaryjny nieaktywny
	bRun:BOOL;						//Zezwolenie na podanie knotów do wbijaków - jak maszyna w Execute musi być na 1
	bRun1: BOOL;					//Zezwolenie na wbicie knota
	bRun2: BOOL;					//Zezwolenie na wbicie knota
	bHoming:BOOL;					//Zezwolenie na wykonanie bazowania i pozycjonowania podajnika
	bHeightSet:BOOL;				//Ustaw wysokość
	bIgnoreError:BOOL;				//Ignorowania błędów cyklu pracy
	bReset:BOOL;					//Reset błędu, jeśli w stanie "eError"
	lrPositionHeightSV:LREAL;		//Wysokość zadana na której ma znajdować się podajnik
	lrMaxHeight:LREAL;				//Maksymalna wysokość podajnika platynek
	lrMinHeight:LREAL;				//Minimalna wysokość podajnika platynek
	bManualMovement:BOOL; 			//Uruchomienie trybu ruchów ręcznych
	
	_SENSORS_:BOOL;	
	bWheelLevelSensor			: BOOL;	
	bWheelSensor				: BOOL;
	bQueFullAfterWheelSensor	: BOOL;			//Czujnik zapełnienia rękawa
	bQueFullSensor				: BOOL;			//Czujnik zapełnienia rękawa
	bWickAtPipe					: BOOL;			//Czujnik na końcu rękawa
	bSeparatorPos1				: BOOL;			//Separator nad torem 1
	bSeparatorPos2				: BOOL;			//Separator nad torem 2
	bQueFullAtSleve1			: BOOL;			//Czujnik zapełnienia rękawa 1
	bQueFullAtSleve2			: BOOL;			//Czujnik zapełnienia rękawa 2
	bWickAtSleve1				: BOOL;			//Czujnik na końcu rękawa 1
	bWickAtSleve2				: BOOL;			//Czujnik na końcu rękawa 2
	bSleve1SeparatorIn			: BOOL;			//Separator pod rękawem
	bSleve1SeparatorOut			: BOOL;			//Separator nad butelką
	bSleve2SeparatorIn			: BOOL;			//Separator pod rękawem
	bSleve2SeparatorOut			: BOOL;			//Separator nad butelką
	bHammer1Up					: BOOL;			//Wbijak pozycja górna
	bHammer1Down				: BOOL;			//Wbijak pozycja dolna
	bHammer2Up					: BOOL;			//Wbijak pozycja górna
	bHammer2Down				: BOOL;			//Wbijak pozycja dolna
	bFormPositioningHide1		: BOOL;			//Wbijak pozycja dolna
	bFormPositioningHide2		: BOOL;			//Wbijak pozycja dolna
	
	_HEIGHTMOTOR_ :BOOL;	
	udiHeightMotorEncoderCV		: UDINT;		//Sygnał impulsów enkodera siłownika
	bHeightEncoderSetCDone		: BOOL;	
	rHeightMotorPositionOffset 	: REAL;			//Wysokość bazowani podnośnika
//	nPositionHeightCV			: LREAL;		//Aktualna wysokość podajnika platynek
	
	_BOWLMOTOR_ :BOOL;
	bEngineOK					: BOOL;					//Wejście czujnika zabezpieczenia silnika 
	InEngineVelocityCV 			: UDINT;		
	InEngineSTW 				: UINT; 				// Statusword transportera wejściowo wyjściowego
	IbEngineWcState				: BOOL; 				// Statusword transportera wejściowo wyjściowego
	_PARAMETERS_:BOOL;
	iTimeDelayOn				: INT; 					//Czas na właczenie silnika sortera po zaniku sygnału przepełnienia z rękawa
	iTimeDelayOff				: INT; 					// Czas na wylączenie silnika sortera po wykryciu sygnału przepełnienia z rękawa sortera
	iTimeToEmptySleeveError		: INT;					// Czas do włączenia alrmu pustego rękawa

	_ALARMINFO_ :BOOL;
	iStationIndex:UDINT;					//Numer stacji 
	sStationName:WSTRING;					//Nazwa stacji	

	
END_VAR
VAR_OUTPUT
	eState: E_Station;						//Stan ogólny bloku
	eRunningStateFeeder: E_WickFeederSorterState;		//Stan podajnika platynek
	eRunningState1: E_WickFeederState;		//Stan podajnika platynek
	eRunningState2: E_WickFeederState;		//Stan podajnika platynek
	
	bError: BOOL;							//Błąd stacji
	nErrorNr: UDINT;						//Nr błędu podajnika platynek
	sErrorDescription:STRING(200);			//Opis błędu
	sErrorDescription2: STRING(200);		//Opis błędu 2
	sErrorStationName:STRING;				//Nazwa stacji
	udiStationID:UDINT;						// Nr stacji
	
	tCycleTime:TIME;	
	bHomingDone:BOOL;						//Wymagane ponowne bazowanie (blad podczas bazowania lub stop awaryjny)	
	bCycleDone1	:BOOL;
	bCycleDone2	:BOOL;
	bCycleNotDone1:BOOL;
	bCycleNotDone2:BOOL;
	
	bHeightMotorUp				:BOOL;					//Sterowanie silnikiem podnośnika  - RUCH W GÓRĘ
	bHeightMotorDown			:BOOL;					//Sterowanie silnikiem podnośnika  - RUCH W DÓŁ
	lrHeightMotorCV				:LREAL;					//Aktualna pozycja podnośnika
	udiHeightMotorEncoderSetCV	: UDINT;		
	bHeightEncoderSetC			: BOOL;					// Zerowanie enkodera
	
	bSorterEngine 				: BOOL; 				// Sterowanie silnikiem sortera
	QnEngineVelocitySV 			: UDINT; 				// Nastawa prędkości
	QnEngineCTW 				: UINT;  				// Controlword transportera we/wy	
	
	bStopper1					: BOOL;			//Stoper1 przed separatorem
	bStopper2					: BOOL;			//Stoper2 przed separatorem
	bSeparator1					: BOOL;			//Separator nad torem 1
	bSeparator2					: BOOL;			//Separator nad torem 2
	bSleve1SeparatorActIn		: BOOL;			//Separator pod rękawem
	bSleve1SeparatorActOut		: BOOL;			//Separator nad butelką
	bSleve2SeparatorActIn		: BOOL;			//Separator pod rękawem
	bSleve2SeparatorActOut		: BOOL;			//Separator nad butelką
	bHammer1					: BOOL;			//Wbijak 
	bHammer2					: BOOL;			//Wbijak
	bFormPositioning			: BOOL;			//Pozycjonowanie 1
	bBlow1						: BOOL;
	bSleeveBlow					: BOOL;
	
	bWarning					: BOOL;
END_VAR

VAR_IN_OUT
	bManualHeightMotorUp		: BOOL;					//Ruch ręczny podnośnika stacji w górę
	bManualHeightMotorDown		: BOOL;					//Ruch ręczny podnośnika stacji w dół
	bManualSorterEngine			: BOOL;					//Ręczne włączenie silnika sortera
	bManualSorterAir			: BOOL;					//Ręczne włączenie zaworu wydmuchu
	
	bManualStopper				: BOOL;		
	bManualStopper2				: BOOL;						
	bManualSeparator1			: BOOL;			//Separator nad torem 1
	bManualSeparator2			: BOOL;			//Separator nad torem 2
	bManualSleve1SeparatorActIn	: BOOL;			//Separator pod rękawem
	bManualSleve1SeparatorActOut: BOOL;			//Separator nad butelką
	bManualSleve2SeparatorActIn	: BOOL;			//Separator pod rękawem
	bManualSleve2SeparatorActOut: BOOL;			//Separator nad butelką
	bManualHammer1				: BOOL;			//Wbijak 
	bManualHammer2				: BOOL;			//Wbijak					
	bManualFormPositioning		: BOOL;			//Wbijak	
END_VAR

VAR
	//Podnośnik Jiesang	
	fbHeightMotorEncoder: FB_JiesangActuatorEncoderModul;	// Blok enkodera podnośnika chwytaka stabilizującego pod zakręcarką	
	bHeightMotorEncoderCounterReset:BOOL; 				//Sygnał resetu enkodera
	bHeightMotorEncoderHomed:BOOL;						//Informacja od enkodera że jest zbazowany
	lrLastPositionHeightCV			: LREAL;			//Pozycja podnośnika w poprzednim cyklu programu
	
	
	fbInverter: FB_MitsubishiInverter;
	tonInverterError: TON;

	
	eLastState: E_Station;							//Stan ogólny bloku
	eLastRunningState: E_WickFeederState;			//Stan podbloku
	eLastStateTemp: E_Station;						//Stan ogólny bloku
	eLastRunningStateTemp: E_WickFeederState;		//Stan podbloku
	bStateError: BOOL;
	tonEstopDelay: TON;
	
	
	
	bManualPositionChanged						: BOOL;
	
	tonHomingSensor								: TON;
	tonHeightNoChange			: TON; 					// Timer wykrycia braku ruchu siłownika zmiany wysokości stacji
	tonHeightNoChangeTime		: TON; 					// Timer wykrycia braku ruchu siłownika zmiany wysokości stacji
	tofHeightMotorDown			: TOF;
	tofHeightMotorUp			: TOF;
	
	tonLimitPosMinReachedDelay	: TON;					// Timer osoiągniecia minimalnej wyskości 
	tonLimitPosMaxReachedDelay	: TON;					// Timer osiągnięcia maksymalnej wyskości
	tonSortingEngineOn			: TON;					// Opóźnienie po załączeniu napędu
	tonSortingEngineOff			: TON;					// Opóźnienie wyłączenia napędu
	tonSleeveFullEngineOn		: TON;					// Czas załączenia napędu po wykrciu braku nasadek
	tonEngineBlocked			: TON;					// Zablokowany silnik	
	tonTryUnblockWheel			: TON;					// Czas ruchu falownika w drugą stronę
	
	tonAirBeforeStart			: TON;					// Czasówka opóźeniani przedmuchu
	tonAirBeforeStart2			: TON;					// Czasówka opóźeniani przedmuchu
	tonAirAfterStop				: TON;					// Czasówka przedmuchu po zatrzymaniu
	tonStoppingTime				: TON;					// Czasówka zbyt długiego zatrzymawania
	
	rtEncoderHomed				: R_TRIG;				// Bit zakończenia enkodera
	rtWheelSensor				: R_TRIG;
	bTryUnblockWheel 			: BOOL;
	iTryUnblockWheel 			: INT;
	
	TimerOn						: TON;
	TimerOff					: TON;
	bImpOn						: BOOL;
	
	tonHammer1Down				: TON;
	tonHammer2Down				: TON;
	
	tonErrorHeightChange		: TON; 					// Timer błędu zacięcia się podnośnika
	tonEmptySleeveError			: TON;					// Timer pustego rękawa
	tonMaxHeightError			: TON;					// Timer ustawienia zbyt dużej wysokości stacji
	tonMinHeightError			: TON;					// Timer ustawienia zbyt małej wysokości stacji
	tonSorterEngineError		: TON;
	tonbSeparatorPos1AndNotbWickAtSleve1 : TON;	
	tonbSeparatorPos2AndNotbWickAtSleve2 : TON;		
	tonbSeparatorPos1 : TON;
	tonbSeparatorPos2 : TON;
	tonbWickAtPipe : TON;
	tobbSleve1SeparatorIn : TON;
	tobbSleve2SeparatorIn : TON;

	tonSeparatorPos1Error		: TON;
	tonSeparatorPos2Error		: TON;
	tonSleve1SeparatorInError	: TON;
	tonSleve1SeparatorOutError	: TON;
	tonSleve2SeparatorInError	: TON;
	tonSleve2SeparatorOutError	: TON;
	tonHammer1UpError			: TON;
	tonHammer1DownError			: TON;
	tonHammer2UpError			: TON;
	tonHammer2DownError			: TON;
	tonWickBlocked1				: TON;
	tonWickBlocked2				: TON;
	
	
	//Zmienne od EVENTLOGGER
	bAlarmInit 						: BOOL := TRUE; 
	nAlarmNumerator					: INT;
	arfbAlarm						: ARRAY[0..19] OF  FB_TcAlarm;		//Tablica bloczków błędów
	fbSourceInfo 					: FB_TcSourceInfo;
	iSourceInfo						: I_TcSourceInfo;
	sAlarmTest						: STRING;
	//Koniec zmiennych od EVENTLOGGER

	rtbSeparator1: R_TRIG;
	rtbSeparator2: R_TRIG;
	rtbSleve1SeparatorActIn: R_TRIG;
	rtbSleve1SeparatorActOut: R_TRIG;
	rtbSleve2SeparatorActIn: R_TRIG;
	rtbSleve2SeparatorActOut: R_TRIG;
	fbbQueFullAtSleve1: FB_InputFilter_v2;
	fbbQueFullAtSleve2: FB_InputFilter_v2;	
	fbbWickAtPipe: FB_InputFilter_v2;
	fbbNotWickAtPipe: FB_InputFilter_v2;	
	iSortingCase: INT;
	tonCaseA: TON;
	tonCaseB: TON;	
	tonCaseC: TON;	
	tonCaseD: TON;
	bSeparatorLast:BOOL;
	bWickBlocked:BOOL;
	tonLowLevelSensor:TON;
END_VAR


ACT_HeightMotor();
ACT_ErrorHandling();
ACT_Warning();
ACT_Inverter();
ACT_Control();
ACT_Signals();
//Statistics();
//EncoderTest();
//aStationID();
(*Zapisywanie ostatniego stanu*)
// IF eLastStateTemp<>eState THEN
// 	eLastState := eLastStateTemp;
// END_IF
// eLastStateTemp := eState;
// IF eLastRunningStateTemp<>eRunningState THEN
// 	eLastRunningState := eLastRunningStateTemp;
// END_IF
// eLastRunningStateTemp := eRunningState;
(*Koniec Zapisywanie ostatniego stanu*)

lrLastPositionHeightCV:=lrHeightMotorCV;

ACTION ACT_Control:
	(*****Wyłączenie enable*****)
	IF NOT bEnable THEN
		IF eState <> E_Station.eDisabled AND eState <> E_Station.ePreparingToDisable THEN
				eState 				:= E_Station.ePreparingToDisable; 
		END_IF	
	END_IF

	(*****Estop*****)
	IF NOT bEstop  THEN	
		IF eState <> E_Station.eAborted AND eState <> E_Station.eAborting AND eState <> E_Station.eDisabled THEN
				eState 				:= E_Station.eAborting; 
		END_IF
	END_IF


	CASE eState OF
//--------------------------------------------------------------------------------
// Stan maszyny po wyłączeniu i przygotowanie do uruchomienia
	E_Station.eDisabled: 					// Stan nieaktywnosci (Stacja wyłączona) 
	
		IF bEnable THEN
			eState 				:= E_Station.ePreparingToReady; 
		END_IF 
		
//--------------------------------------------------------------------------------
// Stan maszyny po zatrzymaniu awaryjnym   
	E_Station.eAborted: 					// Stan bezpiecznego zatrzymania (po Abortingu) 

		IF bEStop THEN
			eState 				:= E_Station.ePreparingToReady;
		END_IF
		
//--------------------------------------------------------------------------------
// Stan maszyny naciśnieciu estopa 	
	E_Station.eAborting:                 	// Stan bezpiecznego zatrzymywania (po EStopie)
// 		bGate1:= FALSE;
// 		bGate2:= FALSE;
	
		ACT_ResetCommands();

		eState 						:=  E_Station.eAborted;  
		//eRunningState				:=	E_LidFeederState.eReady;
		
//--------------------------------------------------------------------------------
// Stan masyzny po wykryciu błędu			
	E_Station.eError:                 	 	// Stan błędu 	
		
		ACT_ResetCommands();
		
		IF bReset THEN
			eState 				:= E_Station.eResetting;
			bError := FALSE;
		END_IF
		
//--------------------------------------------------------------------------------
// Stan masyzny po wykryciu błędu
	E_Station.eResetting:					// Stan resetowania bledu (po Errorze)
// 			CASE udiErrorID-udiStationIndex OF
// 		
// 				//Error 8 - Błąd falownika
// 				9:
// 					fbInverter.bReset	:= TRUE;
// 					bError 				:= FALSE;
// 				ELSE
// 					bError := FALSE;	
// 			END_CASE		
		
		IF NOT bError AND fbInverter.eState = E_Station.eReady THEN
			fbInverter.bReset	:= FALSE;	
			{warning 'Sprawdzić błąd falownika CapFeeder'}
			nErrorNr 			:=	0;
			sErrorDescription 	:=	'';
			eState 				:=	E_Station.ePreparingToReady;
			//eRunningState		:=	E_CapFeederState.eReady;
		ELSE
			eState 				:=	E_Station.eError;
		END_IF
    
//--------------------------------------------------------------------------------
// Stan ruchoow manualnych
	E_Station.eManualMovement:     			// Stan ruchów manualnych  
   
		ACT_ManualMovements();
		IF bManualHeightMotorUp OR bManualHeightMotorDown OR bSeparator1 OR bSeparator2 OR 
			bSleve1SeparatorActIn OR bSleve2SeparatorActIn OR bSleve1SeparatorActOut OR bSleve2SeparatorActOut THEN
				//bManualPositionChanged		:= TRUE;
			END_IF
		//Wyjście z trybu serwisowego
		IF NOT bManualMovement THEN
			
			bHeightMotorUp				:=	FALSE;
			bHeightMotorDown			:=	FALSE;
			bStopper1					:= FALSE;
			bStopper2					:= TRUE;			
 			bSeparator1					:= FALSE;
 			bSeparator2					:= FALSE;
 			bSleve1SeparatorActIn		:= FALSE;  
 			bSleve1SeparatorActOut	    := FALSE;
 			bSleve2SeparatorActIn	    := FALSE;
 			bSleve2SeparatorActOut	    := FALSE;
 			bHammer1				    := FALSE;
 			bHammer2				    := FALSE;
			bBlow1						:= FALSE;
			bSleeveBlow						:= FALSE;
			bFormPositioning			:= FALSE;
			
			IF bManualPositionChanged THEN
				bHomingDone				:= FALSE;
				bManualPositionChanged	:= FALSE;
			END_IF
			
			eState:=E_Station.eReady;
		END_IF
		

//--------------------------------------------------------------------------------
// Stan rozpoczecia bazowania
	E_Station.eHoming:						// Stan bazowania 
		
		ACT_Homing();
		IF NOT bHoming AND NOT bHeightSet THEN
			bHeightMotorDown					:=	FALSE;
			bHeightMotorUp						:=	FALSE;
		   eState								:=E_Station.ePreparingToReady;
		END_IF		
		
//--------------------------------------------------------------------------------
// Stan zakończenia bazowania
	E_Station.eHomingDone:                  // Stan wykonania bazowania 
	
		bHeightMotorDown					:=	FALSE;
		bHeightMotorUp						:=	FALSE;
		//bHeightMotorEncoderCounterReset		:=	FALSE;
		bHomingDone							:=	TRUE;
		IF NOT bHoming AND NOT bHeightSet THEN
		   eState:=E_Station.eReady;
		END_IF
		
//--------------------------------------------------------------------------------
// Stan przygotowania do gotowości
	E_Station.ePreparingToReady:            // Stan przygotowywania do gotowosci (zawsze przed Ready)  
		

		bStopper2							:=	TRUE;		
		bSorterEngine						:=	FALSE;

		eState								:=	E_Station.eReady;	
		eRunningState1						:=	E_WickFeederState.eReady;
		eRunningState2						:=	E_WickFeederState.eReady;		
//-------------------------------------------------------------------------------
// Stan przygotowania do wyłączenia maszyny
	E_Station.ePreparingToDisable:          // Stan przygotowywania do nieaktywnosci (po wyłączeniu Enable) 
		
// 		bGate1:= FALSE;
// 		bGate2:= FALSE;
		bHomingDone									:= FALSE;	
		bSorterEngine:=FALSE;
//		bSorterAir:=FALSE;
		bHeightMotorUp:= NOT tonHomingSensor.Q;
		bHeightMotorDown:=FALSE;	
		IF tonHeightNoChange.Q OR tonHeightNoChangeTime.Q THEN
			bHeightMotorUp			:=	FALSE;
			bHeightMotorDown		:=	FALSE;	
			//eRunningState			:=	E_CapFeederState.eReady;		
			eState					:=	E_Station.eDisabled;
		END_IF	
			
//--------------------------------------------------------------------------------
// Stan gotowości
	E_Station.eReady:						// Stan gotowosci 
	
		IF bRun  THEN
			eState 				:= E_Station.eStarting; 
		END_IF
		IF bHoming OR bHeightSet THEN
			bHomingDone							:=	FALSE;
			eState 								:= E_Station.eHoming; 
		END_IF
		IF bManualMovement THEN
			//Jeśli przejście w tryb ruchów manualnych przepisz wszystkie stany siłowników sterowanych przez moduł
			//aby zapobiec ewentualnym kolizjom po wejściu w tryb serwisowy
			fbInverter.bDirection 		:= TRUE;
		
			bManualPositionChanged		:= FALSE;
			bHeightMotorUp				:= bManualHeightMotorUp;
			 bManualHeightMotorDown		:=	bHeightMotorDown		;
			 bManualSorterEngine        :=	bSorterEngine			;
			 bManualSorterAir           :=	bBlow1					;
			 bManualSorterAir            :=	bSleeveBlow					;
			 bManualStopper                 :=	bStopper1			;	
			 bManualStopper2	                    :=	bStopper2	;			
			 bManualSeparator1			        :=    bSeparator1	;			
			 bManualSeparator2                   :=    bSeparator2	;			
			 bManualSleve1SeparatorActIn         :=    bSleve1SeparatorActIn	;
    		 bManualSleve1SeparatorActOut        :=    bSleve1SeparatorActOut	;
    		 bManualSleve2SeparatorActIn         :=    bSleve2SeparatorActIn	;
    		 bManualSleve2SeparatorActOut        :=    bSleve2SeparatorActOut	;
    		 bManualHammer1                      :=    bHammer1				    ;
    		 bManualHammer2                      :=    bHammer2				    ;
			 bManualFormPositioning             :=	bFormPositioning		    ;
					
			eState 						:= E_Station.eManualMovement; 
		END_IF
		IF NOT bRun THEN
			bCycleDone1 		:= FALSE;
			bCycleNotDone1 		:= FALSE;	
			bCycleDone2 		:= FALSE;
			bCycleNotDone2 		:= FALSE;	
		END_IF
		IF NOT bRun1 THEN
			bCycleDone1 		:= FALSE;
			bCycleNotDone1 		:= FALSE;	
		END_IF	
		IF NOT bRun2 THEN
			bCycleDone2 		:= FALSE;
			bCycleNotDone2 		:= FALSE;	
		END_IF		
//--------------------------------------------------------------------------------
// Stan zatrzymywania
	E_Station.eStopping:					// Stan zatrzymywania 
		
//		bSorterAir 		:= 	TRUE;
		bSorterEngine 	:=	FALSE;
//		IF tonStoppingTime.Q AND eRunningState1=E_WickFeederSorterState.eReady AND eRunningState2=E_WickFeederSorterState.eReady THEN
		IF tonStoppingTime.Q  THEN
			
			ACT_ResetCommands();
			//eRunningState							:= E_CapFeederState.eReady;
			eState									:= E_Station.eReady;
		END_IF

		
//--------------------------------------------------------------------------------
// Stan uruchomienia lini ( po eReady)
	E_Station.eStarting:                  	// Stan uruchamiania (po Ready)
//		iValvesCycleCase		:=0;
		eState					 := E_Station.eRunning; 

//--------------------------------------------------------------------------------
// Stan wykonywania pracy
	E_Station.eRunning:               		// Stan wykonywania cyklu (po Startingu), w tym stanie osobny

		ACT_Running();
		IF NOT bRun THEN 					(*Przerywanie cyklu*)
			eState				:= E_Station.eStopping;
			//bCycleNotDone		:= TRUE;
		END_IF
		(*IF bCycleDone OR bCycleNotDone THEN (*Cykl zakończony*)
			eState 				 := E_Station.eReady;
		END_IF*)						
		
		
END_CASE
END_ACTION

ACTION ACT_ErrorHandling:
(*
Alarm_0620	620	Error	Blokada podnośnika lub brak zasilania - sprawdź czujnik lub odblokuj mechanicznie
Alarm_0621	621	Error	Pusty rękaw sortera - uzupełnij nasadki
Alarm_0622	622	Error	Wartość zadana wysokości jest większa od maksymalnej - zmień ustawienia w recepturze {0}
Alarm_0623	623	Error	Wartość zadana wysokości jest mniejsza od minimalnej - zmień ustawienia w recepturze {0}
Alarm_0624	624	Error	Błąd falownika
Alarm_0625	625	Error	Błąd siłownika rozdzielacza pozycja 1
Alarm_0626	626	Error	Błąd siłownika rozdzielacza pozycja 2
Alarm_0627	627	Error	Błąd wysunięcia siłownika separatora 1
Alarm_0628	628	Error	Błąd cofnięcia siłownika separatora 1
Alarm_0629	629	Error	Błąd wysunięcia siłownika separatora 2
Alarm_0630	630	Error	Błąd cofnięcia siłownika separatora 2
Alarm_0631	631	Error	Błąd wysunięcia wbijaka 1
Alarm_0632	632	Error	Błąd cofnięcia wbijaka 1
Alarm_0633	633	Error	Błąd wysunięcia wbijaka 2
Alarm_0634	634	Error	Błąd cofnięcia wbijaka 2
Alarm_0635	635	Error	Blokada knota w rękawie 1
Alarm_0636	636	Error	Blokada knota w rękawie 2
*)

IF bAlarmInit THEN
    bAlarmInit := FALSE; 
	fbSourceInfo.Clear();
	fbSourceInfo.sName:=wsLiteral_TO_UTF8(sStationName);//'Machine';
	fbSourceInfo.nId:=udiStationID;//2700;
	// Alarm_0620	620	Error	Blokada podnośnika lub brak zasilania - sprawdź czujnik lub odblokuj mechanicznie
    arfbAlarm[0].CreateEx(stEventEntry := TC_EVENTS.AlarmClass.Alarm_0620, bWithConfirmation:= FALSE,  ipSourceInfo:= fbSourceInfo); 
	// Alarm_0621	621	Error	Pusty rękaw sortera - uzupełnij nasadki
	arfbAlarm[1].CreateEx(stEventEntry := TC_EVENTS.AlarmClass.Alarm_0621, bWithConfirmation:= FALSE,  ipSourceInfo:= fbSourceInfo); 
	// Alarm_0622	622	Error	Wartość zadana wysokości jest większa od maksymalnej - zmień ustawienia w recepturze {0}
	arfbAlarm[2].CreateEx(stEventEntry := TC_EVENTS.AlarmClass.Alarm_0622, bWithConfirmation:= FALSE,  ipSourceInfo:= fbSourceInfo); 
	// Alarm_0623	623	Error	Wartość zadana wysokości jest mniejsza od minimalnej - zmień ustawienia w recepturze {0}
	arfbAlarm[3].CreateEx(stEventEntry := TC_EVENTS.AlarmClass.Alarm_0623, bWithConfirmation:= FALSE,  ipSourceInfo:= fbSourceInfo); 
	// Alarm_0624	624	Error	Błąd falownika
	arfbAlarm[4].CreateEx(stEventEntry := TC_EVENTS.AlarmClass.Alarm_0624, bWithConfirmation:= FALSE,  ipSourceInfo:= fbSourceInfo); 
	// Alarm_0625	625	Error	Błąd siłownika rozdzielacza pozycja 1
	arfbAlarm[5].CreateEx(stEventEntry := TC_EVENTS.AlarmClass.Alarm_0625, bWithConfirmation:= FALSE,  ipSourceInfo:= fbSourceInfo); 
	// Alarm_0626	626	Error	Błąd siłownika rozdzielacza pozycja 2
	arfbAlarm[6].CreateEx(stEventEntry := TC_EVENTS.AlarmClass.Alarm_0626, bWithConfirmation:= FALSE,  ipSourceInfo:= fbSourceInfo); 
	// Alarm_0627	627	Error	Błąd wysunięcia siłownika separatora 1
	arfbAlarm[7].CreateEx(stEventEntry := TC_EVENTS.AlarmClass.Alarm_0627, bWithConfirmation:= FALSE,  ipSourceInfo:= fbSourceInfo); 
	// Alarm_0628	628	Error	Błąd cofnięcia siłownika separatora 1
	arfbAlarm[8].CreateEx(stEventEntry := TC_EVENTS.AlarmClass.Alarm_0628, bWithConfirmation:= FALSE,  ipSourceInfo:= fbSourceInfo); 
	// Alarm_0629	629	Error	Błąd wysunięcia siłownika separatora 2
	arfbAlarm[9].CreateEx(stEventEntry := TC_EVENTS.AlarmClass.Alarm_0629, bWithConfirmation:= FALSE,  ipSourceInfo:= fbSourceInfo); 
	// Alarm_0630	630	Error	Błąd cofnięcia siłownika separatora 2
	arfbAlarm[10].CreateEx(stEventEntry := TC_EVENTS.AlarmClass.Alarm_0630, bWithConfirmation:= FALSE,  ipSourceInfo:= fbSourceInfo); 
	// Alarm_0631	631	Error	Błąd wysunięcia wbijaka 1
	arfbAlarm[11].CreateEx(stEventEntry := TC_EVENTS.AlarmClass.Alarm_0631, bWithConfirmation:= FALSE,  ipSourceInfo:= fbSourceInfo);
	// Alarm_0632	632	Error	Błąd cofnięcia wbijaka 1
	arfbAlarm[12].CreateEx(stEventEntry := TC_EVENTS.AlarmClass.Alarm_0632, bWithConfirmation:= FALSE,  ipSourceInfo:= fbSourceInfo);
	// Alarm_0633	633	Error	Błąd wysunięcia wbijaka 2
	arfbAlarm[13].CreateEx(stEventEntry := TC_EVENTS.AlarmClass.Alarm_0633, bWithConfirmation:= FALSE,  ipSourceInfo:= fbSourceInfo);
	// Alarm_0634	634	Error	Błąd cofnięcia wbijaka 2
	arfbAlarm[14].CreateEx(stEventEntry := TC_EVENTS.AlarmClass.Alarm_0634, bWithConfirmation:= FALSE,  ipSourceInfo:= fbSourceInfo);
	// Alarm_0635	635	Error	Blokada knota w rękawie 1
	arfbAlarm[15].CreateEx(stEventEntry := TC_EVENTS.AlarmClass.Alarm_0635, bWithConfirmation:= FALSE,  ipSourceInfo:= fbSourceInfo);
	// Alarm_0636	636	Error	Blokada knota w rękawie 2
	arfbAlarm[16].CreateEx(stEventEntry := TC_EVENTS.AlarmClass.Alarm_0636, bWithConfirmation:= FALSE,  ipSourceInfo:= fbSourceInfo);
END_IF


//OBSŁUGA BŁĘDÓW 
//tonEstopDelay			(IN:=bEstop,	PT:=T#5S); //Opóżnienie po EStopie w celu blokoady błędów, powietrze jest później niż Estop a sygnał z czujnika nie pokazuje braku powietrza bo jest odcinany za tym

//************LISTA BŁĘDÓW***************
bStateError:= (eState=E_Station.eError) OR (eState=E_Station.eResetting);(* OR bIgnoreError; *)
//Error 1 - podnośnik nie porusza się pomimo wysterowania 
tonErrorHeightChange(IN:=(bHeightMotorUp OR bHeightMotorDown) AND lrLastPositionHeightCV=lrHeightMotorCV, PT:=T#3S);
tonEmptySleeveError(IN:=NOT bQueFullSensor AND bRun, PT:=INT_TO_TIME(iTimeToEmptySleeveError)*1000); //Było 30, teraz jest z receptur
tonMaxHeightError(IN:=lrPositionHeightSV>lrMaxHeight AND NOT bHomingDone AND eState=E_Station.eReady,PT:=T#30S);
tonMinHeightError(IN:=lrPositionHeightSV<lrMinHeight AND NOT bHomingDone AND eState=E_Station.eReady,PT:=T#30S);
tonSorterEngineError(IN:= NOT bEngineOK AND bSorterEngine, PT:=T#3S);
tonInverterError(IN:=fbInverter.bError AND NOT bStateError, PT:=T#3S);

IF bEnable THEN
	// Alarm_0620	620	Error	Blokada podnośnika lub brak zasilania - sprawdź czujnik lub odblokuj mechanicznie
	IF tonErrorHeightChange.Q THEN
		IF NOT arfbAlarm[0].bActive THEN
			bHeightMotorUp:=FALSE;
			bHeightMotorDown:=FALSE;
			arfbAlarm[0].Raise(nTimeStamp:=0);
		END_IF
	ELSE	
		IF  arfbAlarm[0].bActive AND bReset THEN
			arfbAlarm[0].Clear(nTimeStamp:=0, bResetConfirmation:= FALSE);
		END_IF
	END_IF
	
	// Alarm_0621	621	Error	Pusty rękaw sortera - uzupełnij nasadki
	IF tonEmptySleeveError.Q THEN
		IF NOT arfbAlarm[1].bActive THEN
			arfbAlarm[1].Raise(nTimeStamp:=0);
		END_IF
	ELSE	
		IF  arfbAlarm[1].bActive AND bReset THEN
			arfbAlarm[1].Clear(nTimeStamp:=0, bResetConfirmation:= FALSE);
		END_IF
	END_IF
	
	// Alarm_0622	622	Error	Wartość zadana wysokości jest większa od maksymalnej - zmień ustawienia w recepturze {0}
	IF tonMaxHeightError.Q THEN
		arfbAlarm[2].ipArguments.Clear() .AddLReal(lrMaxHeight);
		IF NOT arfbAlarm[2].bActive THEN
// 			bHeightMotorUp:=FALSE;
// 			bHeightMotorDown:=FALSE;
			arfbAlarm[2].Raise(nTimeStamp:=0);
		END_IF
	ELSE	
		IF  arfbAlarm[2].bActive AND bReset THEN
			arfbAlarm[2].Clear(nTimeStamp:=0, bResetConfirmation:= FALSE);
		END_IF
	END_IF
	
	// Alarm_0623	623	Error	Wartość zadana wysokości jest mniejsza od minimalnej - zmień ustawienia w recepturze {0}
		IF tonMinHeightError.Q THEN
			arfbAlarm[3].ipArguments.Clear() .AddLReal(lrMinHeight);
		IF NOT arfbAlarm[3].bActive THEN
// 			bHeightMotorUp:=FALSE;
// 			bHeightMotorDown:=FALSE;
			arfbAlarm[3].Raise(nTimeStamp:=0);
		END_IF
	ELSE	
		IF  arfbAlarm[3].bActive AND bReset THEN
			arfbAlarm[3].Clear(nTimeStamp:=0, bResetConfirmation:= FALSE);
		END_IF
	END_IF
	
	// Alarm_0624	624	Error	Błąd falownika
	IF tonInverterError.Q THEN
		IF NOT arfbAlarm[4].bActive THEN
			arfbAlarm[4].Raise(nTimeStamp:=0);
		END_IF
		IF arfbAlarm[4].bActive AND bReset THEN
			fbInverter.bReset := TRUE;
		END_IF
	ELSE	
		IF  arfbAlarm[4].bActive AND bReset THEN
			arfbAlarm[4].Clear(nTimeStamp:=0, bResetConfirmation:= FALSE);
		END_IF
	END_IF			

	// Alarm_0625	625	Error	Błąd siłownika rozdzielacza pozycja 1
	tonSeparatorPos1Error(IN:=(bSeparator1 AND NOT bSeparatorPos1 ),PT:= T#2S(*T#2S*)); 
	IF tonSeparatorPos1Error.Q THEN
		IF NOT arfbAlarm[5].bActive THEN
			bSeparator1:=FALSE;	
			arfbAlarm[5].Raise(nTimeStamp:=0);
		END_IF
	ELSE	
		IF  arfbAlarm[5].bActive AND bReset THEN
			arfbAlarm[5].Clear(nTimeStamp:=0, bResetConfirmation:= FALSE);
		END_IF
	END_IF;
	// Alarm_0626	626	Error	Błąd siłownika rozdzielacza pozycja 2
	tonSeparatorPos2Error(IN:=(bSeparator2 AND NOT bSeparatorPos2 ),PT:= T#2S); 
	IF tonSeparatorPos1Error.Q THEN
		IF NOT arfbAlarm[6].bActive THEN
			bSeparator2:=FALSE;	
			arfbAlarm[6].Raise(nTimeStamp:=0);
		END_IF
	ELSE	
		IF  arfbAlarm[6].bActive AND bReset THEN
			arfbAlarm[6].Clear(nTimeStamp:=0, bResetConfirmation:= FALSE);
		END_IF
	END_IF;	
	// Alarm_0627	627	Error	Błąd wysunięcia siłownika separatora 1
	tonSleve1SeparatorInError(IN:=bSleve1SeparatorActIn AND NOT bSleve1SeparatorIn,PT:= T#2S);	
	IF tonSleve1SeparatorInError.Q THEN
		IF NOT arfbAlarm[7].bActive THEN
			bSleve1SeparatorIn:=FALSE;	
			arfbAlarm[7].Raise(nTimeStamp:=0);
		END_IF
	ELSE	
		IF  arfbAlarm[7].bActive AND bReset THEN
			arfbAlarm[7].Clear(nTimeStamp:=0, bResetConfirmation:= FALSE);
		END_IF
	END_IF;	
	// Alarm_0628	628	Error	Błąd cofnięcia siłownika separatora 1
	tonSleve1SeparatorOutError(IN:=bSleve1SeparatorActOut AND NOT bSleve1SeparatorOut,PT:= T#2S);
	IF tonSleve1SeparatorOutError.Q THEN
		IF NOT arfbAlarm[8].bActive THEN
			bSleve1SeparatorOut:=FALSE;	
			arfbAlarm[8].Raise(nTimeStamp:=0);
		END_IF
	ELSE	
		IF  arfbAlarm[8].bActive AND bReset THEN
			arfbAlarm[8].Clear(nTimeStamp:=0, bResetConfirmation:= FALSE);
		END_IF
	END_IF;
	// Alarm_0629	629	Error	Błąd wysunięcia siłownika separatora 2
	tonSleve2SeparatorInError(IN:=bSleve2SeparatorActIn AND NOT bSleve2SeparatorIn,PT:= T#2S);	
	IF tonSleve2SeparatorInError.Q THEN
		IF NOT arfbAlarm[9].bActive THEN
			bSleve2SeparatorIn:=FALSE;	
			arfbAlarm[9].Raise(nTimeStamp:=0);
		END_IF
	ELSE	
		IF  arfbAlarm[9].bActive AND bReset THEN
			arfbAlarm[9].Clear(nTimeStamp:=0, bResetConfirmation:= FALSE);
		END_IF
	END_IF;	
	// Alarm_0630	630	Error	Błąd cofnięcia siłownika separatora 2
	tonSleve2SeparatorOutError(IN:=bSleve2SeparatorActOut AND NOT bSleve2SeparatorOut,PT:= T#2S);
	IF tonSleve2SeparatorOutError.Q THEN
		IF NOT arfbAlarm[10].bActive THEN
			bSleve2SeparatorOut:=FALSE;	
			arfbAlarm[10].Raise(nTimeStamp:=0);
		END_IF
	ELSE	
		IF  arfbAlarm[10].bActive AND bReset THEN
			arfbAlarm[10].Clear(nTimeStamp:=0, bResetConfirmation:= FALSE);
		END_IF
	END_IF;
	// Alarm_0631	631	Error	Błąd wysunięcia wbijaka 1
	tonHammer1DownError(IN:= bHammer1 AND NOT bHammer1Down ,PT:= T#2S);
	IF tonHammer1DownError.Q THEN
		IF NOT arfbAlarm[11].bActive THEN
			bHammer1:=FALSE;	
			arfbAlarm[11].Raise(nTimeStamp:=0);
		END_IF
	ELSE	
		IF  arfbAlarm[11].bActive AND bReset THEN
			arfbAlarm[11].Clear(nTimeStamp:=0, bResetConfirmation:= FALSE);
		END_IF
	END_IF;
	// Alarm_0632	632	Error	Błąd cofnięcia wbijaka 1
	tonHammer1UpError(IN:= NOT bHammer1 AND NOT bHammer1Up,PT:= T#2S);
	IF tonHammer1UpError.Q THEN
		IF NOT arfbAlarm[12].bActive THEN
			bHammer1:= TRUE;	
			arfbAlarm[12].Raise(nTimeStamp:=0);
		END_IF
	ELSE	
		IF  arfbAlarm[12].bActive AND bReset THEN
			arfbAlarm[12].Clear(nTimeStamp:=0, bResetConfirmation:= FALSE);
		END_IF
	END_IF;
	// Alarm_0633	633	Error	Błąd wysunięcia wbijaka 2
	tonHammer2DownError(IN:= bHammer2 AND NOT bHammer2Down ,PT:= T#2S);
	IF tonHammer2DownError.Q THEN
		IF NOT arfbAlarm[13].bActive THEN
			bHammer2:=FALSE;	
			arfbAlarm[13].Raise(nTimeStamp:=0);
		END_IF
	ELSE	
		IF  arfbAlarm[13].bActive AND bReset THEN
			arfbAlarm[13].Clear(nTimeStamp:=0, bResetConfirmation:= FALSE);
		END_IF
	END_IF;
	// Alarm_0634	634	Error	Błąd cofnięcia wbijaka 2
	tonHammer2UpError(IN:= NOT bHammer2 AND NOT bHammer2Up,PT:= T#2S);
	IF tonHammer2UpError.Q THEN
		IF NOT arfbAlarm[14].bActive THEN
			bHammer2:=TRUE;	
			arfbAlarm[14].Raise(nTimeStamp:=0);
		END_IF
	ELSE	
		IF  arfbAlarm[14].bActive AND bReset THEN
			arfbAlarm[14].Clear(nTimeStamp:=0, bResetConfirmation:= FALSE);
		END_IF
	END_IF;
	// Alarm_0635	635	Error	Blokada knota w rękawie 1
	tonWickBlocked1(IN:=bQueFullAfterWheelSensor AND NOT bQueFullSensor AND bRun, PT:=T#15S);
	IF tonWickBlocked1.Q THEN
		IF NOT arfbAlarm[15].bActive THEN
	
			arfbAlarm[15].Raise(nTimeStamp:=0);
		END_IF
	ELSE	
		IF  arfbAlarm[15].bActive AND bReset THEN
			arfbAlarm[15].Clear(nTimeStamp:=0, bResetConfirmation:= FALSE);
		END_IF
	END_IF;
	// Alarm_0636	636	Error	Blokada knota w rękawie 2
	tonWickBlocked2();
		IF tonWickBlocked2.Q THEN
		IF NOT arfbAlarm[16].bActive THEN
	
			arfbAlarm[16].Raise(nTimeStamp:=0);
		END_IF
	ELSE	
		IF  arfbAlarm[16].bActive AND bReset THEN
			arfbAlarm[16].Clear(nTimeStamp:=0, bResetConfirmation:= FALSE);
		END_IF
	END_IF;


ELSE
		bError 					:= FALSE;
END_IF
//*******KONIEC LISTA BŁĘDÓW***************


//******************PRZEJŚCIE DO eERROR*****************************

IF bError AND NOT bStateError THEN
// 	IF eLastState = eRunning THEN
// 		bCycleNotDone := TRUE;
// 	END_IF
	eState := E_Station.eError;
END_IF

//****************WYŚWIETLANIE STATUSU BLEDU***********************


(*Wyświetlanie błedu na wyjściu*)
bError							:= FALSE;
FOR nAlarmNumerator := 0 TO 19 DO
	bError						:= bError OR arfbAlarm[nAlarmNumerator].bActive;
END_FOR

(*Przepisywanie nazwy stacji*)
//sErrorStationName:=sStationName;



//Jezeli nie zbazowane to potrzebne bazowanie
IF NOT bHeightMotorEncoderHomed  THEN
	bHomingDone:=FALSE;
END_IF
END_ACTION

ACTION ACT_HeightMotor:
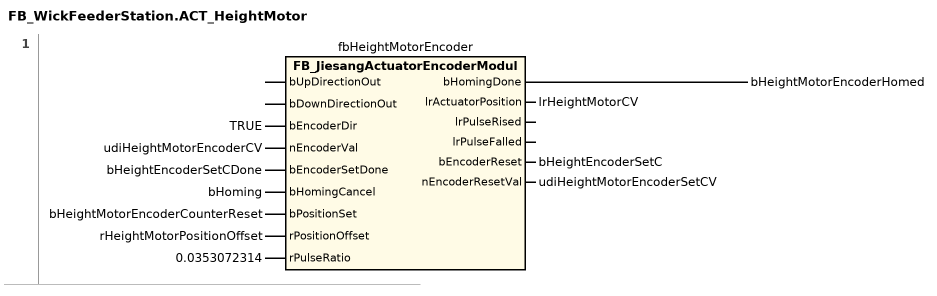
// NETWORK 1
fbHeightMotorEncoder(
    bEncoderDir := TRUE,
    nEncoderVal := udiHeightMotorEncoderCV,
    bEncoderSetDone := bHeightEncoderSetCDone,
    bHomingCancel := bHoming,
    bPositionSet := bHeightMotorEncoderCounterReset,
    rPositionOffset := rHeightMotorPositionOffset,
    rPulseRatio := 0.0353072314,
    lrActuatorPosition => lrHeightMotorCV,
    bEncoderReset => bHeightEncoderSetC,
    nEncoderResetVal => udiHeightMotorEncoderSetCV); // FB_JiesangActuatorEncoderModul
bHeightMotorEncoderHomed := fbHeightMotorEncoder.bHomingDone;
END_ACTION

ACTION ACT_Homing:
//BAZOWANIE

tofHeightMotorDown	(IN:=bHeightMotorDown, PT:=T#1S);	//Zabezpieczenie przed zbyt szybkim przełączeniem pomiędzy Down a Up, bezpiecznieki sie palą
tofHeightMotorUp	(IN:=bHeightMotorUp, PT:=T#1S); 	//Zabezpieczenie przed zbyt szybkim przełączeniem pomiędzy Down a Up, bezpiecznieki sie palą
//Ustaw siłowniki
bStopper1					:= TRUE; //Raczej zablokuj ?
bStopper2					:= TRUE;
//Do zastanowienia
bSeparator1					;
bSeparator2					;
//Podnieś wbijacze
bHammer1					:= FALSE;
bHammer2					:= FALSE;
//Wyłącz odmuchy
bBlow1						:= FALSE;
bSleeveBlow					:= FALSE;
bFormPositioning			:= FALSE;
//Jak wbijacze w górze to ustaw separator na załadunek
IF bHammer1Up THEN
	bSleve1SeparatorActIn	:= TRUE;
	bSleve1SeparatorActOut	:= FALSE;
END_IF

IF bHammer2Up THEN
	bSleve2SeparatorActIn	:= TRUE;
	bSleve2SeparatorActOut	:= FALSE;
END_IF

	
//Podnoszenie stacji do maksymalnej pozycji
IF NOT bHeightMotorEncoderHomed OR rtEncoderHomed.Q THEN
	bHeightMotorUp:= NOT tofHeightMotorDown.Q AND NOT tonHomingSensor.Q;
	bHeightMotorDown:= FALSE;
	IF tonHeightNoChange.Q THEN//OR tonHeightNoChangeTime.Q THEN
		bHeightMotorEncoderCounterReset:=TRUE;
		bHeightMotorUp:=FALSE;
   END_IF
	//Jesli enkoder zbazowany zakończ bazowanie	
	IF rtEncoderHomed.Q  THEN
		bHeightMotorUp:=FALSE;
		bHeightMotorDown:=FALSE;
		eState:=E_Station.eHomingDone;
	END_IF		
		
//Po podniesieniu stacji opuszczanie do ustalonej wysokości
ELSIF bHeightMotorEncoderHomed THEN
	bHeightMotorEncoderCounterReset:=FALSE;
	bHeightMotorUp:=lrHeightMotorCV<=lrPositionHeightSV;
	bHeightMotorDown:=lrHeightMotorCV>=lrPositionHeightSV;
	//Kiedy stacja osiągnie wysokość zadaną
	IF ABS(lrHeightMotorCV-lrPositionHeightSV)<0.5 OR tonLimitPosMaxReachedDelay.Q OR tonLimitPosMinReachedDelay.Q THEN
		bHeightMotorDown:=FALSE;
		bHeightMotorUp:=FALSE;
		//Jak siłowniki na miejscach
		IF bHammer1Up AND bHammer2Up AND bSleve1SeparatorIn AND bSleve2SeparatorIn THEN
			eState:=E_Station.eHomingDone;
		END_IF
	END_IF			
END_IF
END_ACTION

ACTION ACT_Inverter:
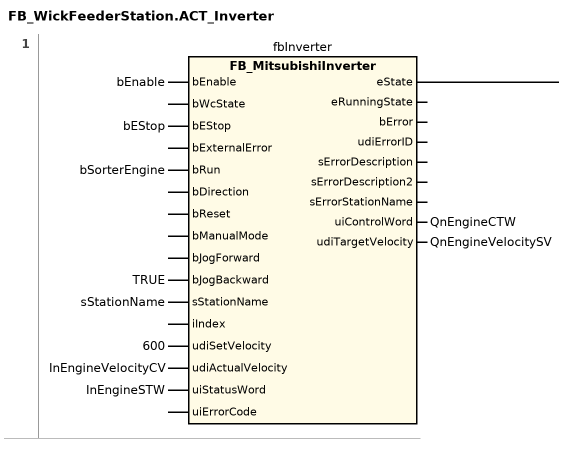
// NETWORK 1
fbInverter(
    bEnable := bEnable,
    bEStop := bEStop,
    bRun := bSorterEngine,
    bJogBackward := TRUE,
    sStationName := sStationName,
    udiSetVelocity := 600,
    udiActualVelocity := InEngineVelocityCV,
    uiStatusWord := InEngineSTW,
    uiControlWord => QnEngineCTW,
    udiTargetVelocity => QnEngineVelocitySV); // FB_MitsubishiInverter
END_ACTION

ACTION ACT_ManualMovements:
//W trybie ruchów manualnych wykonuj ruchy za pomocą rozkazów manualnych

rtbSeparator1				(CLK:=bManualSeparator1				, Q=>);	IF rtbSeparator1.Q				THEN bManualSeparator2				;END_IF	         	
rtbSeparator2				(CLK:=bManualSeparator2				, Q=>);	IF rtbSeparator2.Q				THEN bManualSeparator1			    ;END_IF     
rtbSleve1SeparatorActIn	    (CLK:=bManualSleve1SeparatorActIn	, Q=>);	IF rtbSleve1SeparatorActIn.Q	THEN bManualSleve1SeparatorActOut	;END_IF  
rtbSleve1SeparatorActOut    (CLK:=bManualSleve1SeparatorActOut	, Q=>);	IF rtbSleve1SeparatorActOut.Q 	THEN bManualSleve1SeparatorActIn    ;END_IF
rtbSleve2SeparatorActIn	    (CLK:=bManualSleve2SeparatorActIn	, Q=>);	IF rtbSleve2SeparatorActIn.Q	THEN bManualSleve2SeparatorActOut	;END_IF 
rtbSleve2SeparatorActOut    (CLK:=bManualSleve2SeparatorActOut	, Q=>);	IF rtbSleve2SeparatorActOut.Q 	THEN bManualSleve2SeparatorActIn    ;END_IF



IF NOT bRun THEN
	
	bHeightMotorUp				:= bManualHeightMotorUp;
	bHeightMotorDown			:= bManualHeightMotorDown;
	bSorterEngine				:= bManualSorterEngine;
	bBlow1						:= bManualSorterAir;
	bSleeveBlow					:= bManualSorterAir;
	bStopper1					:= bManualStopper;
	bStopper2					:= bManualStopper2;	
    bSeparator1					:= bManualSeparator1;			
    bSeparator2					:= bManualSeparator2;
    bSleve1SeparatorActIn		:= bManualSleve1SeparatorActIn;    
    bSleve1SeparatorActOut	    := bManualSleve1SeparatorActOut;
    bSleve2SeparatorActIn	    := bManualSleve2SeparatorActIn;
    bSleve2SeparatorActOut	    := bManualSleve2SeparatorActOut;
    bHammer1				    := bManualHammer1;          
    bHammer2				    := bManualHammer2;  
	bFormPositioning			:= bManualFormPositioning;        

END_IF


IF bHoming OR bHeightSet THEN
	eState:=E_Station.eHoming;
END_IF

IF bRun THEN	
	ACT_Running();
END_IF

//Zabezpieczenie przed kolizją stacji poprzez ruch podnośnika	
IF bHeightMotorDown AND lrHeightMotorCV<=lrMinHeight AND NOT bHoming AND NOT bHeightSet THEN
	bHeightMotorDown:=FALSE;
END_IF	

IF bHeightMotorUp AND lrHeightMotorCV>=lrMaxHeight AND NOT bHoming AND NOT bHeightSet THEN
	bHeightMotorUp:=FALSE;
END_IF
END_ACTION

ACTION ACT_ResetCommands:
//Reset komend ruchu 	


			bSorterEngine				:=	FALSE;
			bHeightMotorUp				:=	FALSE;
			bHeightMotorDown			:=	FALSE;
			bStopper1					:= FALSE;
			bStopper2					:= TRUE;			
 			//bSeparator1					:= FALSE;
 			//bSeparator2					:= FALSE;
 			//bSleve1SeparatorActIn		:= FALSE;  
 			//bSleve1SeparatorActOut	    := FALSE;
 			//bSleve2SeparatorActIn	    := FALSE;
 			//bSleve2SeparatorActOut	    := FALSE;
 			bHammer1				    := FALSE;
 			bHammer2				    := FALSE;
			bBlow1						:= FALSE;
			bSleeveBlow					:= FALSE;
			bFormPositioning			:= FALSE;
END_ACTION

ACTION ACT_Running:
//Obsługa sortera knotów - podawanie do separatora
CASE eRunningStateFeeder OF
	
	//NIEGOTOWY
	E_WickFeederSorterState.eDisabled:
		eRunningStateFeeder:=E_WickFeederSorterState.eReady;

	E_WickFeederSorterState.eReady:
		iTryUnblockWheel		:=	0;
		bTryUnblockWheel		:= FALSE;	
		fbInverter.bDirection 	:= TRUE;
		IF bRun THEN
			eRunningStateFeeder			:=E_WickFeederSorterState.eSorting;
		END_IF
	
	E_WickFeederSorterState.eSorting:
		bSorterEngine:=tonAirBeforeStart.Q;
		bBlow1:=TRUE;
		(*Próba odblokowania koła*)
			iTryUnblockWheel := iTryUnblockWheel + 1;
			IF rtWheelSensor.Q THEN
				iTryUnblockWheel	:=	0;
			END_IF
			IF tonEngineBlocked.Q THEN
				bTryUnblockWheel := TRUE;
			END_IF	
			IF bTryUnblockWheel THEN
				fbInverter.bDirection := FALSE;
			END_IF
			IF tonTryUnblockWheel.Q THEN
				iTryUnblockWheel		:=	0;//dp
				bTryUnblockWheel		:= FALSE;
				fbInverter.bDirection 	:= TRUE;
			END_IF

		(* Koniec Podawanie do toru jeden lub dwa*)		
						
		IF tonSortingEngineOff.Q THEN 
			eRunningStateFeeder 			:=E_WickFeederSorterState.eSleeveFull;
		END_IF
	
	E_WickFeederSorterState.eSleeveFull:
		bSorterEngine:=FALSE;
 		bBlow1:=NOT tonAirAfterStop.Q;
		IF tonAirAfterStop.Q THEN
			IF tonSortingEngineOn.Q THEN
				eRunningStateFeeder		:=E_WickFeederSorterState.eSorting; 
			END_IF
		END_IF
	
	E_WickFeederSorterState.eSleeveLowLevel:
		bSorterEngine:=TRUE;
		bBlow1:=TRUE;
		IF tonSortingEngineOff.Q THEN
			eRunningStateFeeder		 	:=E_WickFeederSorterState.eSorting;
		END_IF
	
END_CASE


		(* Koniec Próba odblokowania koła*)		
		CASE iSortingCase OF
			0:
				iSortingCase := iSortingCase	+	10;
				
			10:
				bStopper1:= TRUE;
				bStopper2:= TRUE;
				
				IF	bQueFullSensor THEN
					iSortingCase := iSortingCase	+	10;
				END_IF
				
			20:	
				bStopper1	:= FALSE;
				bStopper2	:= TRUE;
				IF tonCaseA.Q  AND NOT bWickBlocked THEN
					IF NOT fbbQueFullAtSleve1.bOUT AND (NOT bSeparatorLast OR fbbQueFullAtSleve2.bOUT) THEN
							bSeparator1			:= FALSE;
							bSeparator2			:= TRUE;
							IF tonbSeparatorPos2.Q THEN
								iSortingCase := iSortingCase	+	10;
								bSeparatorLast		:= TRUE;
							END_IF
					ELSIF NOT fbbQueFullAtSleve2.bOUT THEN	
							bSeparator1			:= TRUE;
							bSeparator2			:= FALSE;	
							IF tonbSeparatorPos1.Q THEN
								iSortingCase := iSortingCase	+	10;
								bSeparatorLast	:= FALSE;
							END_IF
					END_IF
				ELSIF tonCaseA.Q THEN
					iSortingCase := iSortingCase	+	10;
					bWickBlocked := FALSE;
				END_IF
									
			30:
				iSortingCase := iSortingCase	+	5;

			35:
				bSleeveBlow := TRUE;
				bStopper1	:= TRUE;
				bStopper2	:= FALSE;
				IF tonCaseB.Q AND fbbWickAtPipe.bOUT THEN
					bSleeveBlow  := FALSE;
					iSortingCase := iSortingCase	+	5;
				ELSIF fbbNotWickAtPipe.bOUT THEN
					bSleeveBlow  := FALSE;
					bWickBlocked := TRUE;
					iSortingCase := 10;
				END_IF	
				
			40:
				IF bSeparatorPos1 THEN
						bSeparator1			:= FALSE;
						bSeparator2			:= TRUE;
						iSortingCase		 := iSortingCase	+	10;
				ELSIF bSeparatorPos2 THEN
						bSeparator1			:= TRUE;
						bSeparator2			:= FALSE;		
						iSortingCase	 	:= iSortingCase	+	10;				
				END_IF

			50:	
				IF bSeparator2 AND tonbSeparatorPos2.Q THEN
					iSortingCase	 	:= 0;
				ELSIF bSeparator1 AND tonbSeparatorPos1.Q THEN
					iSortingCase	 	:= 0;				
				END_IF

		END_CASE
		(* Podawanie do toru jeden lub dwa*)


//Obsługa wbijaka 1
CASE eRunningState1 OF
	E_WickFeederState.eDisabled:
		eRunningState1					:= E_WickFeederState.eReady;
	E_WickFeederState.eFilling:
		;
	E_WickFeederState.eReady:	
		IF bWickAtSleve1 AND bRun1 AND NOT bCycleDone1 THEN
			eRunningState1				:= E_WickFeederState.ePuttingWick;
		END_IF
		IF NOT bRun1 THEN
			bCycleDone1 				:= FALSE;
			bCycleNotDone1 				:= FALSE;	
		END_IF
	E_WickFeederState.ePuttingWick:
		bSleve1SeparatorActIn			:= FALSE;			
		bSleve1SeparatorActOut			:= TRUE;
		IF bSleve1SeparatorOut THEN
			bHammer1					:= TRUE;
		END_IF
		//Jak siłownik dojdzie do końca ruchu - DODAĆ czasówkę
		IF tonHammer1Down.Q THEN
			bHammer1					:= FALSE;
			eRunningState1				:= E_WickFeederState.eWickPutted;
		END_IF
		IF NOT bRun1 THEN
			eRunningState1				:= E_WickFeederState.eReady;
		END_IF	
	E_WickFeederState.eWickPutted:
		bCycleDone1:=TRUE;
		IF bHammer1Up THEN
			bSleve1SeparatorActIn		:= TRUE;			
			bSleve1SeparatorActOut		:= FALSE;
			IF tobbSleve1SeparatorIn.Q THEN
				eRunningState1			:= E_WickFeederState.eReady;
			END_IF	
		END_IF
END_CASE	


//Obsługa wbijaka 2
CASE eRunningState2 OF
	E_WickFeederState.eDisabled:
		eRunningState2					:= E_WickFeederState.eReady;
		
	E_WickFeederState.eFilling:
		;
		
	E_WickFeederState.eReady:
		IF bWickAtSleve2 AND bRun2 AND NOT bCycleDone2 THEN
			eRunningState2			:= E_WickFeederState.ePuttingWick;
		END_IF
		IF NOT bRun2 THEN
			bCycleDone2 				:= FALSE;
			bCycleNotDone2 				:= FALSE;	
		END_IF	
		
	E_WickFeederState.ePuttingWick:
		bSleve2SeparatorActIn			:= FALSE;			
		bSleve2SeparatorActOut			:= TRUE;
		IF bSleve2SeparatorOut THEN
			bHammer2					:= TRUE;
		END_IF

		//Jak siłownik dojdzie do końca ruchu - DODAĆ czasówkę
		IF tonHammer2Down.Q  THEN
			bHammer2					:= FALSE;
			eRunningState2				:= E_WickFeederState.eWickPutted;
		END_IF
		IF NOT bRun2 THEN
			eRunningState2				:= E_WickFeederState.eReady;
		END_IF
		
	E_WickFeederState.eWickPutted:
		bCycleDone2:=TRUE;
		IF bHammer2Up THEN
			bSleve2SeparatorActIn		:= TRUE;			
			bSleve2SeparatorActOut		:= FALSE;
			IF tobbSleve2SeparatorIn.Q THEN
				eRunningState2			:= E_WickFeederState.eReady;
			END_IF	
		END_IF
END_CASE
END_ACTION

ACTION ACT_RunningHammer:
		IF bWickAtSleve1 AND bRun1 AND NOT bCycleDone1 THEN
			bSleve1SeparatorActIn		:= FALSE;			
			bSleve1SeparatorActOut		:= TRUE;
			IF bSleve1SeparatorOut THEN
				bHammer1				:= TRUE;
				eRunningState1			:= E_WickFeederState.ePuttingWick;
			END_IF
		END_IF

		IF NOT bRun1 THEN
			bCycleDone1 		:= FALSE;
			bCycleNotDone1 		:= FALSE;	
		END_IF
END_ACTION

ACTION ACT_Signals:
(** Timery na potrzeby bazowania**)
rtEncoderHomed(CLK:=bHeightMotorEncoderHomed,Q=>);
tonHeightNoChange(IN:=((bHeightMotorUp OR bHeightMotorDown OR tonHomingSensor.Q) AND (lrLastPositionHeightCV=lrHeightMotorCV)), PT:=T#2000MS); 
tonLimitPosMinReachedDelay(IN:=(lrHeightMotorCV<=lrMinHeight) AND eState=E_Station.eHoming,PT:=T#2S);
tonLimitPosMaxReachedDelay(IN:=(lrHeightMotorCV>=lrMaxHeight) AND eState=E_Station.eHoming,PT:=T#2S);
	
(** Timery używane podczas pracy stacji**)
tonSortingEngineOff(IN:=((eRunningStateFeeder=E_WickFeederSorterState.eSorting OR eRunningStateFeeder=E_WickFeederSorterState.eSleeveLowLevel) AND bRun AND bQueFullSensor),PT:=INT_TO_TIME(iTimeDelayOff));
tonSortingEngineOn(IN:=((eRunningStateFeeder=E_WickFeederSorterState.eSorting OR eRunningStateFeeder=E_WickFeederSorterState.eSleeveFull) AND bRun AND NOT bQueFullSensor),PT:=INT_TO_TIME(iTimeDelayOn));
tonSleeveFullEngineOn(IN:=(eRunningStateFeeder=E_WickFeederSorterState.eSleeveFull AND bRun AND NOT bQueFullSensor),PT:=INT_TO_TIME(iTimeDelayOff));
rtWheelSensor(CLK:=bWheelSensor, Q=>);
tonEngineBlocked(IN:=iTryUnblockWheel > 1500 AND bSorterEngine AND NOT bTryUnblockWheel,PT:=T#1MS); //Zablokowany silnik
tonTryUnblockWheel(IN:=bTryUnblockWheel, PT:=T#1S900MS);
//tofWickFeederSorterCapSensor(IN:=tonCapFeederSorterCapSensor.Q,PT:=T#100MS); //bylo 200
//tonCapFeederSorterCapSensor(IN:=bSorterCapSensor,PT:=T#3mS);//było 3ms
tonAirBeforeStart(IN:=eRunningStateFeeder=E_WickFeederSorterState.eSorting, PT:=T#1S);
//rtCapFeederSorterCapSensor(CLK:=tofCapFeederSorterCapSensor.Q,Q=>);

